// TwinCAT 3 PLC project CNM_Collections
// Title: CNM_Collections
// Company: ekvip automation GmbH
// Author: tdie
// ProjectVersion: 0.1.1.0
// Description: Concrete Implementations of Collections .. <legal notes> legal notes ================= | SPDX-FileCopyrightText: © 2024 ekvip automation GmbH <info@ekvip.de> | SPDX-License-Identifier: Apache-2.0 | For details check: Apache-2.0_ .. _Apache-2.0: https://www.apache.org/licenses/LICENSE-2.0 .. </legal notes>
// ProgramVersion: 3.1.4026.19
// libraries:
//   CNM_AbstractObject, * (ekvip automation GmbH)
//   CNM_CollectionInterfaces, * (ekvip automation GmbH)
//   CNM_CommandInterfaces, * (ekvip automation GmbH)
//   CNM_CycleManager, * (ekvip automation GmbH)
//   CNM_CycleManagerInterfaces, * (ekvip automation GmbH)
//   CNM_ReturnTypes, * (ekvip automation GmbH)
//   Tc2_System, * (Beckhoff Automation GmbH)
// project tree:
//   Appliers/classes/ ApplierBuilder.TcPOU, ApplierList.TcPOU, ChainedApplier.TcPOU
//   BinaryTree/BBSTIterator/classes/ AbstractBalancedBinarySearchTreeIterator.TcPOU, BfsBbstIterator.TcPOU, DfsBbstIterator.TcPOU, InorderBbstIterator.TcPOU
//   BinaryTree/BBSTIterator/interfaces/Iterator/ IBBSTIterator.TcIO
//   BinaryTree/classes/ BalancedBinarySearchTree.TcPOU, BalancedBinarySearchTreeNode.TcPOU
//   BinaryTree/Set/ InstantSetStrategyExecutor.TcPOU, SetStrategyExecutor.TcPOU
//   BinaryTree/Set/Interfaces/ ISetHelper.TcIO
//   BinaryTree/Tree/ InstantTreeStrategyExecutor.TcPOU, TreeStrategyExecutor.TcPOU
//   BinaryTree/Tree/Interfaces/ ITreeHelper.TcIO
//   Collection/classes/ AbstractCollection.TcPOU, AbstractDisposableContainer.TcPOU, ForEachStrategyExecutor.TcPOU, ForEachInstantStrategyExecutor.TcPOU
//   Factories/classes/ CollectionFactory.TcPOU
//   Iterate/classes/ AbstractIterator.TcPOU
//   Lists/ArrayList/ArrayListIterator/classes/ AbstractArrayListIterator.TcPOU, ForwardArrayListIterator.TcPOU, InverseArrayListIterator.TcPOU
//   Lists/ArrayList/ArrayListIterator/interfaces/Iterator/ IArrayListIterator.TcIO
//   Lists/ArrayList/ArrayListResizingStrategy/ CubicRootResizing.TcPOU, CubicRootUpsizeOnly.TcPOU
//   Lists/ArrayList/ArrayListSorter/ AbstractMergeBasedSorter.TcPOU, ArrayListMergeSorter.TcPOU, ArrayListShellSorter.TcPOU, ArrayListTwinSorter.TcPOU
//   Lists/ArrayList/classes/ ArrayList.TcPOU
//   Lists/ArrayList/ SortingOrder.TcDUT
//   Lists/classes/ AbstractList.TcPOU, SortingStrategyExecutor.TcPOU, InstantSortingStrategyExecutor.TcPOU
//   Lists/ IListHelpers.TcIO
//   Lists/LinkedList/classes/Interfaces/ ILinkedListHelpers.TcIO
//   Lists/LinkedList/classes/LinkedListIterator/classes/ AbstractLinkedListIterator.TcPOU, ForwardLinkedListIterator.TcPOU, InverseLinkedListIterator.TcPOU
//   Lists/LinkedList/classes/LinkedListIterator/interfaces/Iterator/ ILinkedListIterator.TcIO
//   Lists/LinkedList/classes/ DoublyLinkedElement.TcPOU, LinkedList.TcPOU
//   Lists/LinkedList/LinkedListSorter/ LinkedListMergeSorter.TcPOU
//   Lists/Sorter/classes/ AbstractArrayListSorter.TcPOU, AbstractLinkedListSorter.TcPOU, AbstractListSorter.TcPOU
//   Lists/Sorter/classes/Internal/ InvertComparator.TcPOU
//   Lists/Types/ IterationDirection.TcDUT
//   Parameter/ GeneralParameters.TcGVL
//   Project Information/ F_GetCompany.TcPOU, F_GetTitle.TcPOU, F_GetVersion.TcPOU
//   Utils/ FastSwap.TcPOU, log2.TcPOU
//   Version/ Global_Version.TcGVL

// ---- Lists/ArrayList/SortingOrder.TcDUT
{attribute 'qualified_only'}
{attribute 'strict'}
{attribute 'to_string'}
{attribute 'hide'}
TYPE FINAL SortingOrder :
(
	ASCENDING := 0,
	DESCENDING
) SINT;
END_TYPE

// ---- Lists/Types/IterationDirection.TcDUT
(*

## Short summary

This in an enumeration for the iteration direction. It can be forward (position) or backward (negative). 

.. <legal notes>

legal notes
=================
| SPDX-FileCopyrightText: © 2025 ekvip automation GmbH <info@ekvip.de>
| SPDX-License-Identifier: Apache-2.0
| For details check: Apache-2.0_

.. _Apache-2.0: https://www.apache.org/licenses/LICENSE-2.0

.. </legal notes>



*)

{attribute 'qualified_only'}
{attribute 'to_string'}
TYPE IterationDirection :
(
	BACKWARD := -1,
	FORWARD := 1
)DINT := FORWARD;
END_TYPE

// ---- Parameter/GeneralParameters.TcGVL
{attribute 'qualified_only'}
VAR_GLOBAL CONSTANT
	DEFAULT_OPERATIONS_PER_CYCLE :UDINT := 2048;
END_VAR

// ---- Version/Global_Version.TcGVL
{attribute 'TcGenerated'}
{attribute 'no-analysis'}
{attribute 'linkalways'}
// This function has been automatically generated from the project information.
VAR_GLOBAL CONSTANT
	{attribute 'const_non_replaced'}
	stLibVersion_CNM_Collections : ST_LibVersion := (iMajor := 0, iMinor := 1, iBuild := 1, iRevision := 0, nFlags := 0, sVersion := '0.1.1.0');
END_VAR

// ---- BinaryTree/BBSTIterator/interfaces/Iterator/IBBSTIterator.TcIO
(*

## Short summary

This interface extends the IIterator interface for collections by the method attachTree().

.. <legal notes>

legal notes
=================
| SPDX-FileCopyrightText: © 2022 ekvip automation GmbH <info@ekvip.de>
| SPDX-License-Identifier: Apache-2.0
| For details check: Apache-2.0_

.. _Apache-2.0: https://www.apache.org/licenses/LICENSE-2.0

.. </legal notes>

*)

INTERFACE IBBSTIterator EXTENDS CNM_CollectionInterfaces.IIterator

(*

## Short summary

This method attaches an binary balances search tree to the iterator.

.. <legal notes>

legal notes
=================
| SPDX-FileCopyrightText: © 2022 ekvip automation GmbH <info@ekvip.de>
| SPDX-License-Identifier: Apache-2.0
| For details check: Apache-2.0_

.. _Apache-2.0: https://www.apache.org/licenses/LICENSE-2.0

.. </legal notes>


*)

METHOD attachTree 
VAR_INPUT
	(* The tree to be attached, should not be NULL *)
	tree : REFERENCE TO BalancedBinarySearchTree;
END_VAR
END_METHOD

END_INTERFACE

// ---- BinaryTree/Set/Interfaces/ISetHelper.TcIO
INTERFACE INTERNAL ISetHelper EXTENDS CNM_AbstractObject.IObject

(*

## Short summary

Searches an object that is equal to the provided object in terms of the compareTo method (or a comparator provided by the parent).
 
.. <legal notes>

legal notes
=================
| SPDX-FileCopyrightText: © 2023 ekvip automation GmbH <info@ekvip.de>
| SPDX-License-Identifier: Apache-2.0
| For details check: Apache-2.0_

.. _Apache-2.0: https://www.apache.org/licenses/LICENSE-2.0

.. </legal notes>


**Return:** ``TRUE`` when an object that is equal is found, otherwise ``FALSE``

*)

METHOD INTERNAL getEqualObject :BOOL
VAR_INPUT
	(*The object to search for*)
	object 	:CNM_AbstractObject.IObject;
END_VAR
VAR_OUTPUT
	(*The found object or null if not found*)
	foundObject :CNM_AbstractObject.IObject;
END_VAR
END_METHOD

(*

## Short summary

overwrites the content of this set with the intersection of this set and the given set
Set intersection: Common elements between two sets.

**Example:**
Set A = {2, 3, 1, 4}
Set B = {3, 5, 6, 4}

Intersection of A and B: {3, 4}

.. <legal notes>

legal notes
=================
| SPDX-FileCopyrightText: © 2022 ekvip automation GmbH <info@ekvip.de>
| SPDX-License-Identifier: Apache-2.0
| For details check: Apache-2.0_

.. _Apache-2.0: https://www.apache.org/licenses/LICENSE-2.0

.. </legal notes>


**Return:** ``SingleExecutionResult.SUCCESS``: if intersect is complete
	``SingleExecutionResult.ABORTED``: foreign set wasn't valid

*)

METHOD INTERNAL instantIntersect :CNM_ReturnTypes.SingleExecutionResult
VAR_INPUT
	(*foreign set to intersect with*)
	set :CNM_CollectionInterfaces.ISet;
END_VAR
END_METHOD

(*

## Short summary

overwrites the content of this set with the union of this set and the given set
Set union: Combination of all elements from two sets.

**Example:**
Set A = {2, 3, 1, 4}
Set B = {3, 5, 6, 4}

Union of A and B: {1, 2, 3, 4, 5, 6}

.. <legal notes>

legal notes
=================
| SPDX-FileCopyrightText: © 2022 ekvip automation GmbH <info@ekvip.de>
| SPDX-License-Identifier: Apache-2.0
| For details check: Apache-2.0_

.. _Apache-2.0: https://www.apache.org/licenses/LICENSE-2.0

.. </legal notes>


**Return:** ``SUCCESS``: if merge completed
	```SingleExecutionResult.ABORTED``: foreign set wasn't valid

*)

METHOD INTERNAL instantMerge :CNM_ReturnTypes.SingleExecutionResult
VAR_INPUT
	(*foreign set to merge with*)
	set :CNM_CollectionInterfaces.ISet;
END_VAR
END_METHOD

(*

## Short summary

overwrites the content of this set with the set difference of this set and the given set
Set difference: Elements present in one set but not in the other.

**Example:**
Set A = {2, 3, 1, 4}
Set B = {3, 5, 6, 4}

Set difference (A - B): {1, 2}
Set difference (B - A): {5, 6}

.. <legal notes>

legal notes
=================
| SPDX-FileCopyrightText: © 2022 ekvip automation GmbH <info@ekvip.de>
| SPDX-License-Identifier: Apache-2.0
| For details check: Apache-2.0_

.. _Apache-2.0: https://www.apache.org/licenses/LICENSE-2.0

.. </legal notes>


**Return:** ``SingleExecutionResult.SUCCESS``: if insert could made, error if object was already in the tree,
	```SingleExecutionResult.ABORTED``: foreign set wasn't valid

*)

METHOD INTERNAL instantSubtract :CNM_ReturnTypes.SingleExecutionResult
VAR_INPUT
	(*foreign set to construct substraction*)
	set :CNM_CollectionInterfaces.ISet;
END_VAR
END_METHOD

(*

## Short summary

overwrites the content of this set with the intersection of this set and the given set
Set intersection: Common elements between two sets.

**Example:**
Set A = {2, 3, 1, 4}
Set B = {3, 5, 6, 4}

Intersection of A and B: {3, 4}

.. <legal notes>

legal notes
=================
| SPDX-FileCopyrightText: © 2022 ekvip automation GmbH <info@ekvip.de>
| SPDX-License-Identifier: Apache-2.0
| For details check: Apache-2.0_

.. _Apache-2.0: https://www.apache.org/licenses/LICENSE-2.0

.. </legal notes>


**Return:** ``SUCCESS``: if intersect is complete
	``ABORTED``: execute has a falling edge during intersect,
	``BUSY``: Intersect is in Progress
	``ERROR``: the passed collection was not valid / contained invalid Elements

*)

METHOD INTERNAL intersect :CNM_ReturnTypes.SingleExecutionState
VAR_INPUT
	(*foreign set to intersect with*)
	set :CNM_CollectionInterfaces.ISet;
	(*If intersect should be processed*)
	execute		:BOOL;
END_VAR
END_METHOD

(*

## Short summary

overwrites the content of this set with the union of this set and the given set
Set union: Combination of all elements from two sets.

**Example:**
Set A = {2, 3, 1, 4}
Set B = {3, 5, 6, 4}

Union of A and B: {1, 2, 3, 4, 5, 6}

.. <legal notes>

legal notes
=================
| SPDX-FileCopyrightText: © 2022 ekvip automation GmbH <info@ekvip.de>
| SPDX-License-Identifier: Apache-2.0
| For details check: Apache-2.0_

.. _Apache-2.0: https://www.apache.org/licenses/LICENSE-2.0

.. </legal notes>


**Return:** ``SUCCESS``: if merge completed, 
	``ABORTED``: execute has a falling edge during merge,
	``BUSY``: merge is in Progress
	``ERROR``: the passed collection where not valid / contained invalid Elements

*)

METHOD INTERNAL merge :CNM_ReturnTypes.SingleExecutionState
VAR_INPUT
	(*foreign set to merge with*)
	set :CNM_CollectionInterfaces.ISet;
	(*If merge should be processed*)
	execute		:BOOL;
END_VAR
END_METHOD

(*

## Short summary

overwrites the content of this set with the set difference of this set and the given set
Set difference: Elements present in one set but not in the other.

**Example:**
Set A = {2, 3, 1, 4}
Set B = {3, 5, 6, 4}

Set difference (A - B): {1, 2}
Set difference (B - A): {5, 6}

.. <legal notes>

legal notes
=================
| SPDX-FileCopyrightText: © 2022 ekvip automation GmbH <info@ekvip.de>
| SPDX-License-Identifier: Apache-2.0
| For details check: Apache-2.0_

.. _Apache-2.0: https://www.apache.org/licenses/LICENSE-2.0

.. </legal notes>


**Return:** ``SUCCESS``: if insert could made, error if object was already in the tree,
	``ABORTED``: execute has a falling edge during insert,
	``BUSY``: Insert is in Progress
	``ERROR``: the passed collection where not valid / contained invalid Elements

*)

METHOD INTERNAL subtract :CNM_ReturnTypes.SingleExecutionState
VAR_INPUT
	(*foreign set to construct substraction*)
	set :CNM_CollectionInterfaces.ISet;
	(*If substract should be processed*)
	execute		:BOOL;
END_VAR
END_METHOD

END_INTERFACE

// ---- BinaryTree/Tree/Interfaces/ITreeHelper.TcIO
INTERFACE INTERNAL ITreeHelper EXTENDS CNM_AbstractObject.IObject

(*

## Short summary

A method to insert a single element into the tree.

.. <legal notes>

legal notes
=================
| SPDX-FileCopyrightText: © 2022 ekvip automation GmbH <info@ekvip.de>
| SPDX-License-Identifier: Apache-2.0
| For details check: Apache-2.0_

.. _Apache-2.0: https://www.apache.org/licenses/LICENSE-2.0

.. </legal notes>


**Return:** ``SUCCESS``: operation successful
	``ABORTED``: operation was aborted (implementation specific)
	``ERROR``: out of memory

*)

METHOD INTERNAL insert :CNM_ReturnTypes.SingleExecutionResult
VAR_INPUT
	(*the object that should be inserted*)
	object :CNM_AbstractObject.IObject;
END_VAR
END_METHOD

(*

## Short summary

This method inserts all elements of a collection into the tree.

If any value of the collection could not be inserted because of duplication, operation isn't aborted, 
insertion is tried for every element of the collection.

.. <legal notes>

legal notes
=================
| SPDX-FileCopyrightText: © 2025 ekvip automation GmbH <info@ekvip.de>
| SPDX-License-Identifier: Apache-2.0
| For details check: Apache-2.0_

.. _Apache-2.0: https://www.apache.org/licenses/LICENSE-2.0

.. </legal notes>


**Return:** ``SUCCESS``: if insert could be made
	``ABORTED``: execute has a falling edge during insert,
	``BUSY``: Insert is in Progress
	``ERROR``: the passed collection where not valid / contained invalid Elements
	``IDLE``: method was never started

*)

METHOD INTERNAL insertCollection :CNM_ReturnTypes.SingleExecutionState
VAR_INPUT
	(*The collection that should be inserted*)
	collection	:CNM_CollectionInterfaces.ICollection;
	(*If insert should be processed*)
	execute		:BOOL;
END_VAR
END_METHOD

(*

## Short summary

This method inserts all elements of a collection into the tree
This takes only one cycle.

.. <legal notes>

legal notes
=================
| SPDX-FileCopyrightText: © 2022 ekvip automation GmbH <info@ekvip.de>
| SPDX-License-Identifier: Apache-2.0
| For details check: Apache-2.0_

.. _Apache-2.0: https://www.apache.org/licenses/LICENSE-2.0

.. </legal notes>


**Return:** ``SingleExecutionResult.SUCCESS``: operation successful
	``SingleExecutionResult.ERROR``: out of memory
	``SingleExecutionResult.ABORTED``: collection to insert wasn't valid

*)

METHOD INTERNAL instantInsertCollection :CNM_ReturnTypes.SingleExecutionResult
VAR_INPUT
	(*The collection that should be inserted*)
	collection	:CNM_CollectionInterfaces.ICollection;
END_VAR
END_METHOD

(*

## Short summary

Function to remove an object from the tree

.. <legal notes>

legal notes
=================
| SPDX-FileCopyrightText: © 2022 ekvip automation GmbH <info@ekvip.de>
| SPDX-License-Identifier: Apache-2.0
| For details check: Apache-2.0_

.. _Apache-2.0: https://www.apache.org/licenses/LICENSE-2.0

.. </legal notes>


**Return:** ``SUCCESS``: if remove could be made
	``ABORTED``: if object wasn't in the tree
	``ERROR``: if object wasn't valid

*)

METHOD INTERNAL remove :CNM_ReturnTypes.SingleExecutionResult
VAR_INPUT
	(* The object that should be removed *)
	object	:CNM_AbstractObject.IObject;
END_VAR
END_METHOD

END_INTERFACE

// ---- Lists/ArrayList/ArrayListIterator/interfaces/Iterator/IArrayListIterator.TcIO
(*

## Short summary

This interface extends the IIterator interface for collections by the method attachArrayList().

.. <legal notes>

legal notes
=================
| SPDX-FileCopyrightText: © 2022 ekvip automation GmbH <info@ekvip.de>
| SPDX-License-Identifier: Apache-2.0
| For details check: Apache-2.0_

.. _Apache-2.0: https://www.apache.org/licenses/LICENSE-2.0

.. </legal notes>

*)

INTERFACE IArrayListIterator EXTENDS CNM_CollectionInterfaces.IIterator

(*

## Short summary

This method attaches an array list to the iterator.

.. <legal notes>

legal notes
=================
| SPDX-FileCopyrightText: © 2024 ekvip automation GmbH <info@ekvip.de>
| SPDX-License-Identifier: Apache-2.0
| For details check: Apache-2.0_

.. _Apache-2.0: https://www.apache.org/licenses/LICENSE-2.0

.. </legal notes>

*)

METHOD attachArrayList
VAR_INPUT
	(* The list to be attached. Should be a reference of type ``ArrayList`` *)
	list :REFERENCE TO ArrayList;
END_VAR
END_METHOD

END_INTERFACE

// ---- Lists/IListHelpers.TcIO
INTERFACE INTERNAL IListHelpers EXTENDS CNM_CollectionInterfaces.IList

METHOD INTERNAL instantSorting : CNM_ReturnTypes.SingleExecutionResult
VAR_INPUT
	order :SortingOrder;
	(*Optional: the comparator that should be used for the sort. Must not be changed while sort is in process*)
	comparator	: CNM_CollectionInterfaces.CNM_AbstractObject.IComparator := 0;
END_VAR
END_METHOD

PROPERTY INTERNAL listChangeIndex : __XWORD
GET
END_GET
SET
END_SET
END_PROPERTY

METHOD INTERNAL sorting : CNM_ReturnTypes.SingleExecutionState
VAR_INPUT
	execute :BOOL;
	order :SortingOrder;
	(*Optional: the comparator that should be used for the sort. Must not be changed while sort is in process*)
	comparator	: CNM_CollectionInterfaces.CNM_AbstractObject.IComparator := 0;
END_VAR
END_METHOD

END_INTERFACE

// ---- Lists/LinkedList/classes/Interfaces/ILinkedListHelpers.TcIO
INTERFACE INTERNAL ILinkedListHelpers EXTENDS IListHelpers, CNM_CollectionInterfaces.ILinkedList

PROPERTY INTERNAL head : CNM_CollectionInterfaces.IDoublyLinkedElement
GET
END_GET
SET
END_SET
END_PROPERTY

PROPERTY INTERNAL last : CNM_CollectionInterfaces.IDoublyLinkedElement
GET
END_GET
SET
END_SET
END_PROPERTY

END_INTERFACE

// ---- Lists/LinkedList/classes/LinkedListIterator/interfaces/Iterator/ILinkedListIterator.TcIO
(*

## Short summary

This interface extends the IIterator interface for collections by the method attachLinkedList().

.. <legal notes>

legal notes
=================
| SPDX-FileCopyrightText: © 2022 ekvip automation GmbH <info@ekvip.de>
| SPDX-License-Identifier: Apache-2.0
| For details check: Apache-2.0_

.. _Apache-2.0: https://www.apache.org/licenses/LICENSE-2.0

.. </legal notes>

*)

INTERFACE ILinkedListIterator EXTENDS CNM_CollectionInterfaces.IIterator

(*

## Short summary

This method attaches an array list to the iterator.

.. <legal notes>

legal notes
=================
| SPDX-FileCopyrightText: © 2022 ekvip automation GmbH <info@ekvip.de>
| SPDX-License-Identifier: Apache-2.0
| For details check: Apache-2.0_

.. _Apache-2.0: https://www.apache.org/licenses/LICENSE-2.0

.. </legal notes>


**Return:** ``CNM_ReturnTypes.SingleExecutionResult.SUCCESS``: the list could be attached to the iterator

*)

METHOD attachLinkedList : CNM_ReturnTypes.SingleExecutionResult
VAR_INPUT
	(* The list to be attached. Should be of type ``CNM_CollectionInterfaces.ILinkedList`` *)
	list :REFERENCE TO LinkedList;
END_VAR
END_METHOD

END_INTERFACE

// ---- Appliers/classes/ApplierBuilder.TcPOU
FUNCTION_BLOCK ApplierBuilder EXTENDS AbstractDisposableContainer IMPLEMENTS CNM_CollectionInterfaces.IApplierChainBuilder, CNM_CollectionInterfaces.IApplierChainContinue
VAR
	applierList 		:ArrayList;
END_VAR

(*

## Short summary

Method to append another Applier to the chained applier.

.. <legal notes>

legal notes
=================
| SPDX-FileCopyrightText: © 2022 ekvip automation GmbH <info@ekvip.de>
| SPDX-License-Identifier: Apache-2.0
| For details check: Apache-2.0_

.. _Apache-2.0: https://www.apache.org/licenses/LICENSE-2.0

.. </legal notes>


**Return:** ``THIS^```IChainedApplier`

*)


METHOD andThen : CNM_CollectionInterfaces.IApplierChainContinue
VAR_INPUT
	applier :CNM_CollectionInterfaces.IApplier;
END_VAR
THIS^.applierList.append(applier);

andThen := THIS^;
END_METHOD

PROPERTY className : CNM_AbstractObject.ClassName
GET
className := 'ApplierBuilder';
END_GET
END_PROPERTY

(*

## Short summary

This method is called in the destruct method and is intended to zero all references and interfaces that should not be destructed. 
To delete the collection with all its contents, use deepDestruct() instead of destruct().

.. <legal notes>

legal notes
=================
| SPDX-FileCopyrightText: © 2025 ekvip automation GmbH <info@ekvip.de>
| SPDX-License-Identifier: Apache-2.0
| For details check: Apache-2.0_

.. _Apache-2.0: https://www.apache.org/licenses/LICENSE-2.0

.. </legal notes>

*)
METHOD PROTECTED clearContents
THIS^.applierList.clear();
END_METHOD

(*

## Short summary

Mark the object as deleted, as it stays in the memory.

.. <legal notes>

legal notes
=================
| SPDX-FileCopyrightText: © 2022 ekvip automation GmbH <info@ekvip.de>
| SPDX-License-Identifier: Apache-2.0
| For details check: Apache-2.0_

.. _Apache-2.0: https://www.apache.org/licenses/LICENSE-2.0

.. </legal notes>

*)
METHOD FB_Exit : BOOL
VAR_INPUT
	(* TRUE: the exit method is called in order to leave the instance which will be copied afterwards (online change).*)
	bInCopyCode	: BOOL;
END_VAR
IF THIS^.isObjectValid(THIS^.applierList) THEN
	THIS^.applierList.deepDestruct();
END_IF
END_METHOD

METHOD finish : CNM_CollectionInterfaces.IApplier
VAR
	object :CNM_AbstractObject.IObject;
	chainedApplier :POINTER TO ChainedApplier;
	applier1 :CNM_CollectionInterfaces.IApplier; 
	applier2 :CNM_CollectionInterfaces.IApplier; 
	applierNext :CNM_CollectionInterfaces.IApplier; 
END_VAR
IF(THIS^.applierList.size = 1)THEN
	__QUERYINTERFACE(THIS^.applierList.dequeue(), finish);
	THIS^.applierList.clear();
ELSE
	object := THIS^.applierList.dequeue();
	__QUERYINTERFACE(object, applier1);
	object := THIS^.applierList.dequeue();
	__QUERYINTERFACE(object, applier2);
	chainedApplier := __NEW(ChainedApplier(firstApplier := applier1, secondApplier := applier2));
	WHILE(THIS^.applierList.size > 0)DO
	object := THIS^.applierList.dequeue();
		__QUERYINTERFACE(object, applierNext);
		chainedApplier^.andThen(applierNext);
	END_WHILE
	finish := chainedApplier^;
END_IF
END_METHOD

METHOD startWith : CNM_CollectionInterfaces.IApplierChainContinue
VAR_INPUT
	applier :CNM_CollectionInterfaces.IApplier;
END_VAR
THIS^.applierList.clear();
THIS^.applierList.append(applier);

startWith := THIS^;
END_METHOD

END_FUNCTION_BLOCK

// ---- Collection/classes/AbstractDisposableContainer.TcPOU
(*

## Short summary

An abstract class to encapsulate 'destruct','deepDestruct' and 'fb_exit' logic.
'destructContents' must be implemented in the concrete class.

.. <legal notes>

legal notes
=================
| SPDX-FileCopyrightText: © 2025 ekvip automation GmbH <info@ekvip.de>
| SPDX-License-Identifier: Apache-2.0
| For details check: Apache-2.0_

.. _Apache-2.0: https://www.apache.org/licenses/LICENSE-2.0

.. </legal notes>



*)

FUNCTION_BLOCK ABSTRACT AbstractDisposableContainer EXTENDS CNM_AbstractObject.Object

(*

## Short summary

This method is called in the destruct method and is intended to zero all references and interfaces that should not be destructed. 
To delete the collection with all its contents, use deepDestruct() instead of destruct().

.. <legal notes>

legal notes
=================
| SPDX-FileCopyrightText: © 2025 ekvip automation GmbH <info@ekvip.de>
| SPDX-License-Identifier: Apache-2.0
| For details check: Apache-2.0_

.. _Apache-2.0: https://www.apache.org/licenses/LICENSE-2.0

.. </legal notes>

*)

METHOD PROTECTED ABSTRACT clearContents
END_METHOD

(*

## Short summary

This method is a self-destruction if the object was created dynamically.
If the object is a container class, the container content is destroyed with it.

**Attention:** 
	For derivations: **If a derived class needs ``deepDestruct`` this method must be overwritten.**
	otherwise it just calls `Object.destruct`. 


.. <legal notes>

legal notes
=================
| SPDX-FileCopyrightText: © 2022 ekvip automation GmbH <info@ekvip.de>
| SPDX-License-Identifier: Apache-2.0
| For details check: Apache-2.0_

.. _Apache-2.0: https://www.apache.org/licenses/LICENSE-2.0

.. </legal notes>

*)
METHOD deepDestruct
VAR
	(* __DELETE(THIS) is not allowed anymore in Tc 4026.
       tmp is just a helper pointer that points to this instance *)
	tmp : POINTER TO CNM_AbstractObject.Object;
END_VAR
IF (
	Tc2_System.F_CheckMemoryArea(pData := THIS, nSize := SIZEOF(THIS^))
	= Tc2_System.E_TcMemoryArea.Dynamic
) THEN
	tmp := THIS;
	__DELETE(tmp);
END_IF
END_METHOD

(*

## Short summary

This method is a self-destruction if the object was created dynamically.
The disposable container provides the option to clear contents that should not be deleted.

.. <legal notes>

legal notes
=================
| SPDX-FileCopyrightText: © 2025 ekvip automation GmbH <info@ekvip.de>
| SPDX-License-Identifier: Apache-2.0
| For details check: Apache-2.0_

.. _Apache-2.0: https://www.apache.org/licenses/LICENSE-2.0

.. </legal notes>

*)
METHOD FINAL destruct
VAR
	(* __DELETE(THIS) is not allowed anymore in Tc 4026.
       tmp is just a helper pointer that points to this instance *)
	tmp : POINTER TO CNM_AbstractObject.Object;
END_VAR
THIS^.clearContents();
SUPER^.destruct();
END_METHOD

END_FUNCTION_BLOCK

// ---- Appliers/classes/ApplierList.TcPOU
FUNCTION_BLOCK ApplierList 
EXTENDS AbstractDisposableContainer 
IMPLEMENTS CNM_CollectionInterfaces.IApplierList
VAR
	myList 				:ArrayList;
END_VAR

METHOD addApplier : CNM_ReturnTypes.SingleExecutionResult
VAR_INPUT
	applier :CNM_CollectionInterfaces.IApplier;
END_VAR
addApplier := THIS^.myList.append(applier);
END_METHOD

METHOD addAppliers : CNM_ReturnTypes.SingleExecutionResult
VAR_INPUT
	appliers :CNM_CollectionInterfaces.ICollection;
END_VAR
addAppliers := THIS^.myList.appendCollection(appliers);
END_METHOD

PROPERTY className : CNM_AbstractObject.ClassName
GET
className := 'ApplierList';
END_GET
END_PROPERTY

METHOD clear : BOOL
VAR_INPUT
END_VAR
THIS^.myList.clear();
END_METHOD

(*

## Short summary

This method is called in the destruct method and is intended to zero all references and interfaces that should not be destructed. 
To delete the collection with all its contents, use deepDestruct() instead of destruct().

.. <legal notes>

legal notes
=================
| SPDX-FileCopyrightText: © 2025 ekvip automation GmbH <info@ekvip.de>
| SPDX-License-Identifier: Apache-2.0
| For details check: Apache-2.0_

.. _Apache-2.0: https://www.apache.org/licenses/LICENSE-2.0

.. </legal notes>

*)
METHOD PROTECTED clearContents
THIS^.myList.clear();
END_METHOD

(*

## Short summary

This property returns the amount of appliers in the list

.. <legal notes>

legal notes
=================
| SPDX-FileCopyrightText: © 2024 ekvip automation GmbH <info@ekvip.de>
| SPDX-License-Identifier: Apache-2.0
| For details check: Apache-2.0_

.. _Apache-2.0: https://www.apache.org/licenses/LICENSE-2.0

.. </legal notes>

*)

PROPERTY count :UDINT
GET
count := THIS^.myList.size;
END_GET
END_PROPERTY

(*

## Short summary

Mark the object as deleted, as it staiys in the memory.

.. <legal notes>

legal notes
=================
| SPDX-FileCopyrightText: © 2022 ekvip automation GmbH <info@ekvip.de>
| SPDX-License-Identifier: Apache-2.0
| For details check: Apache-2.0_

.. _Apache-2.0: https://www.apache.org/licenses/LICENSE-2.0

.. </legal notes>

*)
METHOD FB_Exit : BOOL
VAR_INPUT
	(* TRUE: the exit method is called in order to leave the instance which will be copied afterwards (online change).*)
	bInCopyCode	: BOOL;
END_VAR
IF THIS^.isObjectValid(THIS^.myList) THEN
	THIS^.myList.deepDestruct();
END_IF
END_METHOD

(*

## Short summary

A method to get an applier at the given index.

.. <legal notes>

legal notes
=================
| SPDX-FileCopyrightText: © 2022 ekvip automation GmbH <info@ekvip.de>
| SPDX-License-Identifier: Apache-2.0
| For details check: Apache-2.0_

.. _Apache-2.0: https://www.apache.org/licenses/LICENSE-2.0

.. </legal notes>


**Return:** CNM_ReturnTypes.ExecutionState

*)

METHOD getApplier : CNM_CollectionInterfaces.IApplier
VAR_INPUT
	index	:UDINT;
END_VAR
VAR
	obj :CNM_AbstractObject.IObject;
END_VAR
THIS^.myList.getObjectAt(index := index, object => obj);
__TRY
	__QUERYINTERFACE(obj, getApplier);
__CATCH
	;
__ENDTRY
END_METHOD

PROPERTY list : CNM_CollectionInterfaces.IArrayList
GET
list := this^.myList;
END_GET
END_PROPERTY

END_FUNCTION_BLOCK

// ---- Lists/ArrayList/classes/ArrayList.TcPOU
(*

## Short summary

Implementation of IArrayList.
Does not allow null objects as data! Object is not null if isObjectValid is true.
Efficient if size stays small and index operations need to be performed in O(1).

**Warning:**
	Calling __DELETE directly on a Collection will bypass the destruct Context and therefore also delete the contained elements.

.. <legal notes>

legal notes
=================
| SPDX-FileCopyrightText: © 2022 ekvip automation GmbH <info@ekvip.de>
| SPDX-License-Identifier: Apache-2.0
| For details check: Apache-2.0_

.. _Apache-2.0: https://www.apache.org/licenses/LICENSE-2.0

.. </legal notes>



*)

{attribute 'enable_dynamic_creation'}
FUNCTION_BLOCK ArrayList EXTENDS AbstractList IMPLEMENTS CNM_CollectionInterfaces.IArrayList
VAR
	(*the container where the elements are stored*)
	container					:POINTER TO CNM_AbstractObject.IObject;
	(*how many space does the container has, NOT how many places are currently taken*)
	currentContainerCapacity	:UDINT;
	(*the sorter used to sort the list*) 
	injectedSorter				:CNM_CollectionInterfaces.IArrayListSorter;
	(*true if the sorter was created inside this list, false if set from outside*)
	privateSorter				:BOOL;
	(* injected resizing strategy *)
	injectedResizingStrategy :CNM_CollectionInterfaces.IResizingStrategy;
END_VAR

(*

## Short summary

This method is called every time the list changes and can notify other components.

.. <legal notes>

legal notes
=================
| SPDX-FileCopyrightText: © 2025 ekvip automation GmbH <info@ekvip.de>
| SPDX-License-Identifier: Apache-2.0
| For details check: Apache-2.0_

.. _Apache-2.0: https://www.apache.org/licenses/LICENSE-2.0

.. </legal notes>



*)

METHOD PROTECTED announceListChange
THIS^.changesToCollection := THIS^.changesToCollection+1;
END_METHOD

(*

## Short summary

This method adds the given object to the end of the list.
Adding NULL-Objects or THIS^ to the list is not possible.

.. <legal notes>

legal notes
=================
| SPDX-FileCopyrightText: © 2022 ekvip automation GmbH <info@ekvip.de>
| SPDX-License-Identifier: Apache-2.0
| For details check: Apache-2.0_

.. _Apache-2.0: https://www.apache.org/licenses/LICENSE-2.0

.. </legal notes>


**Return:** ``CNM_ReturnTypes.SingleExecutionResult.SUCCESS``: new Container could be allocated and data was copied
	``CNM_ReturnTypes.SingleExecutionResult.ERROR``: new Container couldn't be allocated, container left unchanged
	``CNM_ReturnTypes.SingleExecutionResult.ABORTED``: NULL object or the list itself was passed
	
*)
METHOD append :CNM_ReturnTypes.SingleExecutionResult
VAR_INPUT
	(*The object to be appended*)
	object	:CNM_AbstractObject.IObject;
END_VAR
append := CNM_ReturnTypes.SingleExecutionResult.ABORTED;
RETURN(THIS^.isEqual(object) OR_ELSE THIS^.isObjectNull(object));

append :=  THIS^.upscaleContainer(1); 
RETURN(append <> CNM_ReturnTypes.SingleExecutionResult.SUCCESS);
THIS^.container[THIS^.size] := object;
THIS^.incrementSize();
THIS^.announceListChange();
END_METHOD

(*

## Short summary

This method adds all elements of the given collection to the end of this list.

.. <legal notes>

legal notes
=================
| SPDX-FileCopyrightText: © 2025 ekvip automation GmbH <info@ekvip.de>
| SPDX-License-Identifier: Apache-2.0
| For details check: Apache-2.0_

.. _Apache-2.0: https://www.apache.org/licenses/LICENSE-2.0

.. </legal notes>


**Return:** ``CNM_ReturnTypes.SingleExecutionResult.SUCCESS``: new Container not needed / could be allocated and data was copied
	``CNM_ReturnTypes.SingleExecutionResult.ERROR``: new Container couldn't be allocated, container left unchanged
	``CNM_ReturnTypes.SingleExecutionResult.ABORTED``: NULL object or the list itself was passed

*)

METHOD appendCollection :CNM_ReturnTypes.SingleExecutionResult
VAR_INPUT
	(*The collection to be appended*)
	collectionToAppend		:CNM_CollectionInterfaces.ICollection;
END_VAR
VAR
	currentIndex 			:UDINT := 0;
	currentObject 			:CNM_AbstractObject.IObject;
	iterator				:CNM_CollectionInterfaces.IIterator;
	arrayListToAppend		:POINTER TO ArrayList;
	newContainer			:POINTER TO CNM_AbstractObject.IObject;
	newContainerSize 		:UDINT;
END_VAR
VAR CONSTANT
	REGISTER_SIZE :UDINT := SIZEOF(__XWORD);
END_VAR
appendCollection := CNM_ReturnTypes.SingleExecutionResult.ABORTED;
RETURN(THIS^.isObjectNull(collectionToAppend) OR_ELSE THIS^.isEqual(collectionToAppend));
appendCollection := CNM_ReturnTypes.SingleExecutionResult.SUCCESS;
RETURN (collectionToAppend.size = 0);
appendCollection := CNM_ReturnTypes.SingleExecutionResult.ERROR;
THIS^.resizingStrategy.getUpscaledCapacity(requestedSize := THIS^.size + collectionToAppend.size, currentCapacity := THIS^.currentContainerCapacity, newCapacity => newContainerSize);
newContainer := __NEW(__XWORD, newContainerSize);
RETURN(newContainer = 0);
IF (THIS^.size > 0) AND_THEN (Tc2_System.MEMMOVE(newContainer, THIS^.container, THIS^.size * REGISTER_SIZE) = 0) THEN
	__DELETE(newContainer);
	RETURN;
END_IF
IF (__QUERYPOINTER(collectionToAppend, arrayListToAppend)) THEN
	IF (Tc2_System.MEMMOVE(ADR(newContainer[THIS^.size]), arrayListToAppend^.container, collectionToAppend.size*REGISTER_SIZE) = 0) THEN
		__DELETE(newContainer);
		RETURN;
	END_IF
ELSE
	IF (collectionToAppend.createNewIterator(iterator => iterator) <> CNM_ReturnTypes.SingleExecutionResult.SUCCESS) THEN
		__DELETE(newContainer); 
		RETURN;
	END_IF
	
	iterator.iterate(execute := FALSE);
	WHILE (
		iterator.iterate(execute := TRUE, object => currentObject) 
		= CNM_ReturnTypes.SingleExecutionState.BUSY
	) DO
		newContainer[THIS^.size + currentIndex] := currentObject;
		currentIndex := (currentIndex + 1);
	END_WHILE
	iterator.destruct();
	IF (currentIndex < collectionToAppend.size) THEN
		__DELETE(newContainer); 
		RETURN;
	END_IF
END_IF
__DELETE(THIS^.container);
THIS^.container := newContainer;
THIS^.currentContainerCapacity := newContainerSize;
THIS^.incrementSize(collectionToAppend.size);
THIS^.announceListChange();
appendCollection := CNM_ReturnTypes.SingleExecutionResult.SUCCESS;
END_METHOD

(*

## Short summary

This abstract property returns the class name of the concrete object, 
which is useful to check the class name for ``__DELETE``.

.. <legal notes>

legal notes
=================
| SPDX-FileCopyrightText: © 2022 ekvip automation GmbH <info@ekvip.de>
| SPDX-License-Identifier: Apache-2.0
| For details check: Apache-2.0_

.. _Apache-2.0: https://www.apache.org/licenses/LICENSE-2.0

.. </legal notes>

*)
PROPERTY className : CNM_AbstractObject.ClassName
GET
className := 'CNM_Collections.ArrayList';
END_GET
END_PROPERTY

(*

## Short summary

This method clears/deletes all clearable data from this object.

.. <legal notes>

legal notes
=================
| SPDX-FileCopyrightText: © 2022 ekvip automation GmbH <info@ekvip.de>
| SPDX-License-Identifier: Apache-2.0
| For details check: Apache-2.0_

.. _Apache-2.0: https://www.apache.org/licenses/LICENSE-2.0

.. </legal notes>



*)

METHOD clear
__DELETE(THIS^.container);
THIS^.container := __NEW(__XWORD, 10);	

THIS^.collectionSize := 0;
THIS^.currentContainerCapacity := 10;
END_METHOD

(*

## Short summary

This method is called in the destruct method and is intended to zero all references and interfaces that should not be destructed. 
To delete the collection with all its contents, use deepDestruct() instead of destruct().

.. <legal notes>

legal notes
=================
| SPDX-FileCopyrightText: © 2025 ekvip automation GmbH <info@ekvip.de>
| SPDX-License-Identifier: Apache-2.0
| For details check: Apache-2.0_

.. _Apache-2.0: https://www.apache.org/licenses/LICENSE-2.0

.. </legal notes>

*)

METHOD PROTECTED clearContents
VAR CONSTANT
	(* NULL is a constant which is always 0 *)
	NULL				:__XWORD := 0;
END_VAR
Tc2_System.MEMSET(THIS^.container, 0, THIS^.size * SIZEOF(__XWORD));
THIS^.injectedSorter := 0;
THIS^.injectedResizingStrategy := 0;
END_METHOD

(*

## Short summary

This method is used to create a new instance
of the object which has the same internal state as the object.
If the object is a container class, the references to the content objects
are not cloned for this there is the method `ICloneable.deepClone`.

If an object does not support cloning the return value is
``CNM_ReturnTypes.CloneResult.CLONE_IS_NOT_SUPPORTED``.

If there is not enough memory or the cloning fails because the
attribute enable dynamic creation was forgotten the return value is 
``CNM_ReturnTypes.CloneResult.FAILED``.

Only if the return value is ``CNM_ReturnTypes.CloneResult.SUCCESS``
the output ``clonedObject`` points to the new object
otherwise ``clonedObject`` is NULL.  

**Attention:** 
	For derivations: **If a derived class needs ``clone`` this method must be overwritten.**
	and don't forget the attribute ``{attribute 'enable_dynamic_creation'}``  

.. <legal notes>

legal notes
=================
| SPDX-FileCopyrightText: © 2022 ekvip automation GmbH <info@ekvip.de>
| SPDX-License-Identifier: Apache-2.0
| For details check: Apache-2.0_

.. _Apache-2.0: https://www.apache.org/licenses/LICENSE-2.0

.. </legal notes>


**Return:**``CNM_ReturnTypes.CloneResult.SUCCESS``: new object clone was created,
``CNM_ReturnTypes.CloneResult.FAILED``: object clone failed
``CNM_ReturnTypes.CloneResult.CLONE_IS_NOT_SUPPORTED``: object does not support cloning

*)
METHOD clone : CNM_AbstractObject.CNM_ReturnTypes.CloneResult
VAR_OUTPUT
	(* new object instance or NULL if somthing went wrong *)
	clonedObject	:CNM_AbstractObject.IObject;
END_VAR
VAR
	result :CNM_ReturnTypes.SingleExecutionResult;
	miniMe :POINTER TO ArrayList;
END_VAR
clone := CNM_ReturnTypes.CloneResult.FAILED;
miniMe := __NEW(ArrayList);
RETURN (miniMe = 0);
clone := CNM_ReturnTypes.CloneResult.SUCCESS;
clonedObject := miniMe^;
IF (miniMe^.appendCollection(THIS^) <> CNM_ReturnTypes.SingleExecutionResult.SUCCESS) THEN
	clonedObject.destruct();
	clone := CNM_ReturnTypes.CloneResult.FAILED;
	clonedObject := 0;
END_IF
END_METHOD

(*

## Short summary

This method returns a NEW Iterator instance which can iterate the collection.
These iterators can be used parallel independend of each other on the same collection.

**Warning:**
The returned Iterator was created using the __NEW operator and must be destructed to avoid memory leaks!



.. <legal notes>

legal notes
=================
| SPDX-FileCopyrightText: © 2024 ekvip automation GmbH <info@ekvip.de>
| SPDX-License-Identifier: Apache-2.0
| For details check: Apache-2.0_

.. _Apache-2.0: https://www.apache.org/licenses/LICENSE-2.0

.. </legal notes>



*)

METHOD createNewIterator :CNM_CollectionInterfaces.CNM_ReturnTypes.SingleExecutionResult
VAR_OUTPUT
	(*The new created iterator or null if allocation fails *)
	iterator	:CNM_CollectionInterfaces.IIterator;
END_VAR
VAR
	newIterator :POINTER TO ForwardArrayListIterator;
END_VAR
newIterator := __NEW(ForwardArrayListIterator(arrayList := THIS^));
IF (newIterator = 0) THEN
	createNewIterator := CNM_ReturnTypes.SingleExecutionResult.ERROR;
	RETURN;
END_IF
createNewIterator := CNM_ReturnTypes.SingleExecutionResult.SUCCESS;
iterator := newIterator^;
END_METHOD

(*

## Short summary

reduces the collection size by the number of removed elements.

.. <legal notes>

legal notes
=================
| SPDX-FileCopyrightText: © 2025 ekvip automation GmbH <info@ekvip.de>
| SPDX-License-Identifier: Apache-2.0
| For details check: Apache-2.0_

.. _Apache-2.0: https://www.apache.org/licenses/LICENSE-2.0

.. </legal notes>

*)

METHOD PROTECTED decrementSize
VAR_INPUT
	numberOfRemovedElements :UDINT := 1;
END_VAR
THIS^.collectionSize := THIS^.collectionSize - numberOfRemovedElements;
END_METHOD

(*

## Short summary

This method is used to create a new instance
of the object which has the same internal state as the object.
If the object is a container class, the references to the content objects
are cloned too.

If an object does not support cloning the return value is
``CNM_ReturnTypes.CloneResult.CLONE_IS_NOT_SUPPORTED``.

If there is not enough memory or the cloning fails because the
attribute enable dynamic creation was forgotten the return value is 
``CNM_ReturnTypes.CloneResult.FAILED``.
If something goes wrong, then this method must clean up everything
that has been cloned and free the memory again.
**The deepClone either works completely, or not at all**

Only if the return value is ``CNM_ReturnTypes.CloneResult.SUCCESS``
the output ``clonedObject`` points to the new object
otherwise ``clonedObject`` is NULL.  

**Attention:** 
	For derivations: **If a derived class needs ``deepClone`` this method must be overwritten.**
	and don't forget the attribute ``{attribute 'enable_dynamic_creation'}``, even for container content 

.. <legal notes>

legal notes
=================
| SPDX-FileCopyrightText: © 2022 ekvip automation GmbH <info@ekvip.de>
| SPDX-License-Identifier: Apache-2.0
| For details check: Apache-2.0_

.. _Apache-2.0: https://www.apache.org/licenses/LICENSE-2.0

.. </legal notes>


**Return:**``CNM_ReturnTypes.CloneResult.SUCCESS``: new object clone was created,
``CNM_ReturnTypes.CloneResult.FAILED``: object clone failed
``CNM_ReturnTypes.CloneResult.CLONE_IS_NOT_SUPPORTED``: object does not support deep cloning

*)
METHOD deepClone : CNM_AbstractObject.CNM_ReturnTypes.CloneResult
VAR_OUTPUT
	(* new object instance or NULL if somthing went wrong *)
	clonedObject	: CNM_AbstractObject.IObject;
END_VAR
VAR
	result :CNM_ReturnTypes.SingleExecutionResult;
	miniMe :POINTER TO ArrayList;
	newInstance :CNM_CollectionInterfaces.IArrayList;
	clonedSorter :CNM_CollectionInterfaces.IArrayListSorter;
	clonedSorterObject :CNM_AbstractObject.IObject;
	index :UDINT;
	target :UDINT;
	tmpObject :CNM_AbstractObject.IObject;
	currentObject :CNM_AbstractObject.IObject;
END_VAR
deepClone := CNM_ReturnTypes.CloneResult.FAILED;
miniMe := __NEW(ArrayList);
RETURN (miniMe = 0);
deepClone := CNM_ReturnTypes.CloneResult.SUCCESS;
clonedObject := miniMe^;
newInstance := miniMe^;
IF (THIS^.size > 0) THEN
	target := THIS^.size - 1;
	FOR index := 0 TO target DO
		currentObject := THIS^.container[index];
		IF NOT THIS^.isObjectValid(currentObject) THEN
			deepClone := CNM_ReturnTypes.CloneResult.FAILED;
			miniMe^.deepDestruct();
			clonedObject := 0;
			RETURN;
		ELSE 
			deepClone := currentObject.deepClone(clonedObject => tmpObject);
			IF (deepClone <> CNM_ReturnTypes.CloneResult.SUCCESS) THEN 
				miniMe^.deepDestruct();
				clonedObject := 0;
				RETURN;
			END_IF
			IF (miniMe^.append(tmpObject) <> CNM_ReturnTypes.SingleExecutionResult.SUCCESS) THEN
				deepClone := CNM_ReturnTypes.CloneResult.FAILED;
				miniMe^.deepDestruct();
				clonedObject := 0;
				RETURN;
			END_IF
		END_IF
	END_FOR
END_IF
	
RETURN (THIS^.isObjectNull(THIS^.injectedSorter));
THIS^.injectedSorter.deepClone(clonedObject => clonedSorterObject);
__QUERYINTERFACE(clonedSorterObject, clonedSorter);
deepClone := SEL(
	THIS^.isObjectValid(clonedSorter),
	CNM_ReturnTypes.CloneResult.FAILED,
	CNM_ReturnTypes.CloneResult.SUCCESS
);

IF (THIS^.isObjectNull(clonedSorter)) THEN
	deepClone := CNM_ReturnTypes.CloneResult.FAILED;
	miniMe^.deepDestruct();
	clonedObject := 0;
	RETURN;
END_IF
newInstance.setSorter(sorter := clonedSorter);
END_METHOD

(*

## Short summary

This property returns the first object in the list and removes it from the list. 
Can be seen as opposite of prepend.
**Example:**
On a list: (Head -->) A B C, list.dequeue will return A.
**Example 2:**
If you call prepend(x), a dequeue right after will return x.

.. <legal notes>

legal notes
=================
| SPDX-FileCopyrightText: © 2022 ekvip automation GmbH <info@ekvip.de>
| SPDX-License-Identifier: Apache-2.0
| For details check: Apache-2.0_

.. _Apache-2.0: https://www.apache.org/licenses/LICENSE-2.0

.. </legal notes>



*)

METHOD dequeue :CNM_AbstractObject.IObject
VAR CONSTANT
	NULL_REFERENCE :__XWORD := 0;
END_VAR
IF (THIS^.size = 0) THEN
	dequeue := NULL_REFERENCE;
	RETURN;
END_IF
dequeue := THIS^.container[0];
THIS^.leftShiftObjects(1);
THIS^.decrementSize();
THIS^.downscaleContainer();
THIS^.announceListChange();
END_METHOD

(*

## Short summary

This method is called in the deepDestruct method and is intended to destruct all contained Objects of the collection. 
To delete only the collection without deleting all its contents, use destruct() instead of deepDestruct().

.. <legal notes>

legal notes
=================
| SPDX-FileCopyrightText: © 2025 ekvip automation GmbH <info@ekvip.de>
| SPDX-License-Identifier: Apache-2.0
| For details check: Apache-2.0_

.. _Apache-2.0: https://www.apache.org/licenses/LICENSE-2.0

.. </legal notes>

*)

METHOD PROTECTED destructContents
VAR
	currentIndex	:__XWORD;
END_VAR
IF (container <> 0) THEN
	FOR currentIndex := 0 TO (THIS^.currentContainerCapacity - 1) DO
		IF THIS^.isObjectValid(THIS^.container[currentIndex]) THEN
			THIS^.container[currentIndex].deepDestruct();
		END_IF
	END_FOR
END_IF
END_METHOD

(*

## Short summary

This method decreases the container capacity by the current decrease strategy amount.

.. <legal notes>

legal notes
=================
| SPDX-FileCopyrightText: © 2025 ekvip automation GmbH <info@ekvip.de>
| SPDX-License-Identifier: Apache-2.0
| For details check: Apache-2.0_

.. _Apache-2.0: https://www.apache.org/licenses/LICENSE-2.0

.. </legal notes>


**Return:** ``CNM_ReturnTypes.SingleExecutionResult.SUCCESS``: new Container could be allocated and data was copied
	``CNM_ReturnTypes.SingleExecutionResult.ERROR``: new Container couldn't be allocated, container left unchanged

*)

{info 'add logging if containeralloc fails'}
METHOD PROTECTED downscaleContainer :CNM_ReturnTypes.SingleExecutionResult;
VAR
	newContainer 			:POINTER TO CNM_AbstractObject.IObject;
	lastContainerCapacity	:UDINT;
	newContainerCapacity	:UDINT;
END_VAR
IF THIS^.resizingStrategy.getDownscaledCapacity(
		requestedSize := THIS^.size,
		currentCapacity := THIS^.currentContainerCapacity,
		newCapacity => newContainerCapacity
	)
THEN
	newContainer := __NEW(__XWORD, newContainerCapacity);
	IF (newContainer <> 0) THEN
		IF (THIS^.container <> 0) THEN 
			IF (THIS^.size > 0) THEN
				Tc2_System.MEMCPY(newContainer, THIS^.container,  THIS^.size * SIZEOF(__XWORD));
			END_IF
			__DELETE(THIS^.container);
		END_IF
		THIS^.container := newContainer;
		downscaleContainer := CNM_ReturnTypes.SingleExecutionResult.SUCCESS;
	ELSE
		THIS^.currentContainerCapacity := lastContainerCapacity;
		downscaleContainer := CNM_ReturnTypes.SingleExecutionResult.ERROR;
	END_IF
END_IF
END_METHOD

(*

## Short summary

Mark the object as deleted, as it staiys in the memory.

.. <legal notes>

legal notes
=================
| SPDX-FileCopyrightText: © 2022 ekvip automation GmbH <info@ekvip.de>
| SPDX-License-Identifier: Apache-2.0
| For details check: Apache-2.0_

.. _Apache-2.0: https://www.apache.org/licenses/LICENSE-2.0

.. </legal notes>

*)
METHOD FB_Exit : BOOL
VAR_INPUT
	(* TRUE: the exit method is called in order to leave the instance which will be copied afterwards (online change).*)
	bInCopyCode	: BOOL;
END_VAR
VAR
	currentIndex	:__XWORD;
END_VAR
IF (container <> 0) THEN
	FOR currentIndex := 0 TO (THIS^.currentContainerCapacity - 1) DO
		IF THIS^.isObjectValid(THIS^.container[currentIndex]) THEN
			THIS^.container[currentIndex].deepDestruct();
		END_IF
	END_FOR
END_IF
IF (THIS^.container <> 0) THEN
	__DELETE(container);
END_IF
IF THIS^.isObjectValid(THIS^.injectedSorter) THEN
	 THIS^.injectedSorter.deepDestruct();
END_IF
IF THIS^.isObjectValid(THIS^.injectedResizingStrategy) THEN
	THIS^.injectedResizingStrategy.deepDestruct();
END_IF
END_METHOD

(*

## Short summary

This method returns the index of the first object that is equal to the given object.

.. <legal notes>

legal notes
=================
| SPDX-FileCopyrightText: © 2022 ekvip automation GmbH <info@ekvip.de>
| SPDX-License-Identifier: Apache-2.0
| For details check: Apache-2.0_

.. _Apache-2.0: https://www.apache.org/licenses/LICENSE-2.0

.. </legal notes>


**Return:** ``CNM_ReturnTypes.SingleExecutionResult.SUCCESS``: Element was found inside the list
	``CNM_ReturnTypes.SingleExecutionResult.ERROR``: object could not be found in the list
	
*)

METHOD getIndexOf : CNM_ReturnTypes.SingleExecutionResult
VAR_INPUT
	(*the object to get the index from*)
	object	:CNM_AbstractObject.IObject;
END_VAR
VAR_OUTPUT
	(*The index where the first occurence was found, only valid if return value was SUCCESS, else undefined(UDINT#FFFF_FFFF) *)
	index	:UDINT;
END_VAR
VAR
	currentObject 	:CNM_AbstractObject.IObject;
END_VAR
THIS^.iterate(FALSE);
IF (THIS^.isObjectValid(object)) THEN
	WHILE (
		THIS^.iterate(execute := TRUE, object => currentObject) 
		= CNM_ReturnTypes.SingleExecutionState.BUSY
	) DO
		IF (object.isEqual(currentObject)) THEN
			getIndexOf := CNM_ReturnTypes.SingleExecutionResult.SUCCESS;
			RETURN;
		END_IF
		index := index +1;
	END_WHILE
END_IF

//in case of not found set index to UDINT max 
index := UDINT#16#FFFF_FFFF;
getIndexOf := CNM_ReturnTypes.SingleExecutionResult.ERROR;
END_METHOD

(*

## Short summary

This method returns the object at the given index.

.. <legal notes>

legal notes
=================
| SPDX-FileCopyrightText: © 2022 ekvip automation GmbH <info@ekvip.de>
| SPDX-License-Identifier: Apache-2.0
| For details check: Apache-2.0_

.. _Apache-2.0: https://www.apache.org/licenses/LICENSE-2.0

.. </legal notes>


**Return:** ``CNM_ReturnTypes.SingleExecutionResult.SUCCESS``: index within valid range, object could be retrieved
	``CNM_ReturnTypes.SingleExecutionResult.ERROR``: index was out of valid range

*)

METHOD getObjectAt : CNM_ReturnTypes.SingleExecutionResult
VAR_INPUT
	(*the index to access the object from*)
	index	:UDINT;
END_VAR
VAR_OUTPUT
	(*The object found at the index, undefined if ERROR*)
	object	: CNM_AbstractObject.IObject;
END_VAR
VAR CONSTANT
	NULL_REFERENCE :__XWORD := 0;
END_VAR
IF (index >= THIS^.size) THEN
	getObjectAt := CNM_ReturnTypes.SingleExecutionResult.ERROR;
	object := NULL_REFERENCE;
	RETURN;
END_IF

getObjectAt := CNM_ReturnTypes.SingleExecutionResult.SUCCESS;
object := THIS^.container[index];
END_METHOD

(*

## Short summary

Increments the collectionsize by given amount. 

.. <legal notes>

legal notes
=================
| SPDX-FileCopyrightText: © 2025 ekvip automation GmbH <info@ekvip.de>
| SPDX-License-Identifier: Apache-2.0
| For details check: Apache-2.0_

.. _Apache-2.0: https://www.apache.org/licenses/LICENSE-2.0

.. </legal notes>

*)

METHOD PROTECTED incrementSize
VAR_INPUT
	numberOfAddedElements :UDINT := 1;
END_VAR
THIS^.collectionSize := (THIS^.collectionSize + numberOfAddedElements);
END_METHOD

(*

## Short summary

This method inserts the given object at the given index. 
The element that was on this index before is not deleted,
but instead is shifted right by one position together 
with the other elements on indices larger than ``index``.
If ``object`` is not valid, list is left unchanged.

.. <legal notes>

legal notes
=================
| SPDX-FileCopyrightText: © 2022 ekvip automation GmbH <info@ekvip.de>
| SPDX-License-Identifier: Apache-2.0
| For details check: Apache-2.0_

.. _Apache-2.0: https://www.apache.org/licenses/LICENSE-2.0

.. </legal notes>


**Return:** ``CNM_ReturnTypes.SingleExecutionResult.SUCCESS``: insert was successful
	``CNM_ReturnTypes.SingleExecutionResult.ERROR``: insert failed, because container needs to increase but no memory left or index is not in valid range
	``CNM_ReturnTypes.SingleExecutionResult.ABORTED``: NULL object or the list itself was passed
*)

METHOD insertObjectAt :CNM_ReturnTypes.SingleExecutionResult
VAR_INPUT
	(*the index to insert the object at*)
	index	:UDINT;
	(*the object to be inserted*)
	object	:CNM_AbstractObject.IObject;
END_VAR
insertObjectAt := CNM_ReturnTypes.SingleExecutionResult.ABORTED;
RETURN(THIS^.isObjectNull(object) OR_ELSE THIS^.isEqual(object));
insertObjectAt := CNM_ReturnTypes.SingleExecutionResult.ERROR;
RETURN (index > THIS^.size);

IF THIS^.isObjectValid(object) THEN
	THIS^.upscaleContainer(1);
	IF (THIS^.rightShiftObjects(index) <> CNM_ReturnTypes.SingleExecutionResult.SUCCESS) THEN
		THIS^.downscaleContainer();
		RETURN;
	END_IF
	THIS^.container[index] := object;
	THIS^.incrementSize();
	THIS^.announceListChange();
	insertObjectAt := CNM_ReturnTypes.SingleExecutionResult.SUCCESS;
END_IF
END_METHOD

METHOD INTERNAL instantSorting : CNM_ReturnTypes.SingleExecutionResult
VAR_INPUT
	order :SortingOrder;
	(*Optional: the comparator that should be used for the sort. Must not be changed while sort is in process*)
	comparator	: CNM_CollectionInterfaces.CNM_AbstractObject.IComparator := 0;
END_VAR
CASE order OF
SortingOrder.ASCENDING:
	instantSorting := THIS^.sorter.instantSort(
		size := THIS^.size, 
		comparator := comparator, 
		container := THIS^.container, 
		currentListVersion := THIS^.changesToCollection
	);

SortingOrder.DESCENDING:
	instantSorting	:= THIS^.sorter.instantInverseSort(
		size := THIS^.size, 
		container := THIS^.container, 
		currentListVersion := THIS^.changesToCollection
	);
	
END_CASE
END_METHOD


(*

## Short summary

Inverts the order of the elements inside the list. 
Does not apply any kind of sorting, only reverses the elements in the list.

.. <legal notes>

legal notes
=================
| SPDX-FileCopyrightText: © 2022 ekvip automation GmbH <info@ekvip.de>
| SPDX-License-Identifier: Apache-2.0
| For details check: Apache-2.0_

.. _Apache-2.0: https://www.apache.org/licenses/LICENSE-2.0

.. </legal notes>

*)

METHOD invert
VAR
	firstElement	:UDINT := 0;
	lastElement		:UDINT := THIS^.size - 1;
	midLower		:UDINT;
	midUpper		:UDINT;
	loop			:UDINT;
END_VAR
VAR CONSTANT
	REGISTER_SIZE :__XWORD := SIZEOF(__XWORD);
END_VAR
CASE (THIS^.size) OF
0,1: RETURN;
2,3: FastSwap(ADR(THIS^.container[firstElement]), ADR(THIS^.container[lastElement]));RETURN;
ELSE
	loop := SHR(THIS^.size, 1);
	midLower := loop - 1;
	midUpper := THIS^.size - loop;
	
	IF ((loop AND 1) <> 0) THEN
		FastSwap(ADR(THIS^.container[midLower]), ADR(THIS^.container[midUpper]));
		loop := loop - 1;
		midLower := midLower - 1;
		midUpper := midupper + 1;
	END_IF;
	
	loop := MAX(SHR(loop, 1), 1);	
END_CASE
	
REPEAT
	FastSwap(ADR(THIS^.container[firstElement]),ADR(THIS^.container[lastElement]));	
	FastSwap(ADR(THIS^.container[midLower]),ADR(THIS^.container[midUpper]));	
	midLower := midLower - 1;
	midUpper := midupper + 1;
	firstElement := firstElement + 1;
	lastElement := lastElement - 1; 
	loop := loop - 1;
UNTIL (loop = 0) END_REPEAT
END_METHOD

(*

## Short summary

This method returns the next object in the list and returns an execution state.

.. <legal notes>

legal notes
=================
| SPDX-FileCopyrightText: © 2022 ekvip automation GmbH <info@ekvip.de>
| SPDX-License-Identifier: Apache-2.0
| For details check: Apache-2.0_

.. _Apache-2.0: https://www.apache.org/licenses/LICENSE-2.0

.. </legal notes>


**Return:** ``SUCCESS``: if last object from collection was returned,
	``ABORTED``: execute has a falling edge during iterate,
	``BUSY``: When iterate had rising edge on execute and not all objects had been returned yet
	``IDLE``: iterate not in progress, execute is false and iterate reseted 

*)
METHOD PROTECTED iterate :CNM_ReturnTypes.SingleExecutionState
VAR_INPUT
	(*False to init, True to retrieve next element*)
	execute	: BOOL;
END_VAR
VAR_OUTPUT
	(*The current element of the iteration*)
	object	:CNM_AbstractObject.IObject;
END_VAR
VAR_INST
	lastExecute 	:BOOL;
	state 			:CNM_ReturnTypes.SingleExecutionState := CNM_ReturnTypes.SingleExecutionState.IDLE;
	currentIndex	:UDINT;
	cycleManager 	:CNM_CycleManager.SimpleCycleManager;
	currentListVersion :__XWORD;
END_VAR
VAR CONSTANT
	IS_NOT_REFERENCED 	:__XWORD := 0;	
	INIT 		:DINT := CNM_ReturnTypes.DefaultSteps.STEP.INIT;
	ITERATING 	:DINT := INIT +1;
	ERROR 		:DINT := CNM_ReturnTypes.DefaultSteps.STEP.ERROR;
END_VAR
IF (cycleManager.step.current > INIT) THEN
	cycleManager.assert.bitNumber.x.valueIsEqualTo(
		currentValue := currentListVersion,
		expectedValue := THIS^.changesToCollection,
		message := 'This instance of ArrayList has changed between iterate calls'
	);
END_IF

cycleManager(execute := execute);
CASE cycleManager.step.current OF
INIT:
	object := IS_NOT_REFERENCED;
	currentIndex := 0;
	currentListVersion := THIS^.changesToCollection;
	IF (currentIndex < THIS^.size) THEN
		object := THIS^.container[currentIndex];
		currentIndex := currentIndex + 1;
		cycleManager.proceed();
	ELSE
		cycleManager.proceedWith(CNM_ReturnTypes.DefaultSteps.STEP.SUCCESS);
		object := IS_NOT_REFERENCED;
	END_IF
ITERATING:
	IF (currentIndex < THIS^.size) THEN
		object := THIS^.container[currentIndex];
		currentIndex := currentIndex + 1;
	ELSE
		cycleManager.proceedWith(CNM_ReturnTypes.DefaultSteps.STEP.SUCCESS);
		object := IS_NOT_REFERENCED;
	END_IF
ERROR:
	object := IS_NOT_REFERENCED;
END_CASE

iterate := cycleManager.state;
END_METHOD

(*

## Short summary

This method shifts the data in the container to the left at the given index.
It memsets the free created gap at the end of the container.
leftShift(0) : A B C D -> B C D
leftShift(1) : A B C D -> A C D
leftShift(1, 2) : A B C D -> A D

.. <legal notes>

legal notes
=================
| SPDX-FileCopyrightText: © 2025 ekvip automation GmbH <info@ekvip.de>
| SPDX-License-Identifier: Apache-2.0
| For details check: Apache-2.0_

.. _Apache-2.0: https://www.apache.org/licenses/LICENSE-2.0

.. </legal notes>


**Return:** ``CNM_ReturnTypes.SingleExecutionResult.SUCCESS``: leftshift was successful
	``CNM_ReturnTypes.SingleExecutionResult.ERROR``: startindex was either zero ,less than distance or greater thansize, distance greater than size

*)

METHOD PROTECTED leftShiftObjects :CNM_ReturnTypes.SingleExecutionResult;
VAR_INPUT
	(*where the leftshift should start, position of the first element which will shift to the left. All elements after this are also shifted by the same amount.*)
	startIndex :UDINT;
	(* the size of the gap to be shifted to the left as IObjects *)
	distance :UDINT := 1;
END_VAR
VAR
	objectsToShift :UDINT;
END_VAR
VAR CONSTANT
	IS_NOT_REFERENCED 	:USINT := 0;
	REGISTER_SIZE :UDINT := SIZEOF(__XWORD);
END_VAR
leftShiftObjects := CNM_ReturnTypes.SingleExecutionResult.ERROR;
RETURN((distance >= THIS^.size) OR_ELSE (startIndex = 0) OR_ELSE (startIndex < distance) OR_ELSE (THIS^.size < startIndex));
objectsToShift := THIS^.size - startIndex;
Tc2_System.MEMMOVE(ADR(THIS^.container[startIndex-distance]), ADR(THIS^.container[startIndex]), objectsToShift * REGISTER_SIZE);
Tc2_System.MEMSET(ADR(THIS^.container[THIS^.size-distance]), IS_NOT_REFERENCED, distance * REGISTER_SIZE);
leftShiftObjects := CNM_ReturnTypes.SingleExecutionResult.SUCCESS;
END_METHOD

(*

## Short summary

This property returns the last object in the list and removes it from the list. 
Can be seen as opposite of append.
**Example:**
On a list: (Head -->) A B C, list.pop will return C.
**Example 2:**
If you call append(x), a pop right after will return x.

.. <legal notes>

legal notes
=================
| SPDX-FileCopyrightText: © 2022 ekvip automation GmbH <info@ekvip.de>
| SPDX-License-Identifier: Apache-2.0
| For details check: Apache-2.0_

.. _Apache-2.0: https://www.apache.org/licenses/LICENSE-2.0

.. </legal notes>



*)

METHOD pop :CNM_AbstractObject.IObject
VAR CONSTANT
	NULL_REFERENCE :__XWORD := 0;
END_VAR
IF (THIS^.size = 0) THEN
	pop := NULL_REFERENCE;
	RETURN;
END_IF
pop := THIS^.container[THIS^.size-1];
THIS^.container[THIS^.size-1] := NULL_REFERENCE;
THIS^.decrementSize();
THIS^.downscaleContainer();
THIS^.announceListChange();
END_METHOD

(*

## Short summary

This method adds the given object to the start of the list.
Adding NULL-Objects or THIS^ to the list is not possible.

.. <legal notes>

legal notes
=================
| SPDX-FileCopyrightText: © 2022 ekvip automation GmbH <info@ekvip.de>
| SPDX-License-Identifier: Apache-2.0
| For details check: Apache-2.0_

.. _Apache-2.0: https://www.apache.org/licenses/LICENSE-2.0

.. </legal notes>


**Return:** ``CNM_ReturnTypes.SingleExecutionResult.SUCCESS``: new Container not needed / could be allocated and data was copied
	``CNM_ReturnTypes.SingleExecutionResult.ERROR``: new Container couldn't be allocated, container left unchanged
	``CNM_ReturnTypes.SingleExecutionResult.ABORTED``: NULL object or the list itself was passed
*)
METHOD prepend :CNM_ReturnTypes.SingleExecutionResult
VAR_INPUT
	(*The object to be prepended*)
	object	: CNM_AbstractObject.IObject;
END_VAR
prepend := THIS^.insertObjectAt(index := 0, object := object);
END_METHOD

(*

## Short summary

This method adds all elements of the given collection to the start of this list. 
The order is given by the default iterator of the given collection.
If the collection to prepend is null or contains no element, list is unchanged.

.. <legal notes>

legal notes
=================
| SPDX-FileCopyrightText: © 2025 ekvip automation GmbH <info@ekvip.de>
| SPDX-License-Identifier: Apache-2.0
| For details check: Apache-2.0_

.. _Apache-2.0: https://www.apache.org/licenses/LICENSE-2.0

.. </legal notes>


**Return:** ``CNM_ReturnTypes.SingleExecutionResult.SUCCESS``: prepend was successful
	``CNM_ReturnTypes.SingleExecutionResult.ERROR``: collection to prepend didn't fit in old container, and new container couldn't be allocated
	``CNM_ReturnTypes.SingleExecutionResult.ABORTED``: NULL object or this arraylist was passed
	
*)
METHOD prependCollection :CNM_ReturnTypes.SingleExecutionResult
VAR_INPUT
	(*The collection to be prepended*)
	collectionToPrepend		:CNM_CollectionInterfaces.ICollection;
END_VAR
VAR
	currentIndex 			:UDINT;
	currentObject 			:CNM_AbstractObject.IObject;
	offset 					:__UXINT;
	iterator				:CNM_CollectionInterfaces.IIterator;
	newContainer			:POINTER TO CNM_AbstractObject.IObject;
	arrayListToPrepend		:POINTER TO ArrayList;
	newContainerSize		:UDINT;
END_VAR
VAR CONSTANT
	REGISTER_SIZE :UDINT := SIZEOF(__XWORD);
END_VAR
prependCollection := CNM_ReturnTypes.SingleExecutionResult.ABORTED;
RETURN(THIS^.isObjectNull(collectionToPrepend) OR_ELSE THIS^.isEqual(collectionToPrepend));
prependCollection := CNM_ReturnTypes.SingleExecutionResult.SUCCESS;
RETURN (collectionToPrepend.size = 0);
prependCollection := CNM_ReturnTypes.SingleExecutionResult.ERROR;
THIS^.resizingStrategy.getUpscaledCapacity(requestedSize := THIS^.size + collectionToPrepend.size, currentCapacity := THIS^.currentContainerCapacity, newCapacity => newContainerSize);
newContainer := __NEW(__XWORD, newContainerSize);
RETURN(newContainer = 0);
IF (Tc2_System.MEMMOVE(ADR(newContainer[collectionToPrepend.size]), THIS^.container, THIS^.size * REGISTER_SIZE) = 0) THEN
	__DELETE(newContainer);
	RETURN;
END_IF
IF (__QUERYPOINTER(collectionToPrepend, arrayListToPrepend)) THEN
	IF (Tc2_System.MEMMOVE(newContainer, arrayListToPrepend^.container, collectionToPrepend.size*REGISTER_SIZE) = 0) THEN
		__DELETE(newContainer);
		RETURN;
	END_IF
ELSE
	IF (collectionToPrepend.createNewIterator(iterator => iterator) <> CNM_ReturnTypes.SingleExecutionResult.SUCCESS) THEN
		__DELETE(newContainer); 
		RETURN;
	END_IF
	
	iterator.iterate(execute := FALSE);
	WHILE (
		iterator.iterate(execute := TRUE, object => currentObject) 
		= CNM_ReturnTypes.SingleExecutionState.BUSY
	) DO
		newContainer[currentIndex] := currentObject;
		currentIndex := (currentIndex + 1);
	END_WHILE
	iterator.destruct();
	IF (currentIndex < collectionToPrepend.size) THEN
		__DELETE(newContainer); 
		RETURN;
	END_IF
END_IF
__DELETE(THIS^.container);
THIS^.container := newContainer;
THIS^.currentContainerCapacity := newContainerSize;
THIS^.incrementSize(collectionToPrepend.size);
THIS^.announceListChange();
prependCollection := CNM_ReturnTypes.SingleExecutionResult.SUCCESS;
END_METHOD

(*

## Short summary

This method removes the first instance of the given object from the list.
Passing a null object leaves the list unchanged.

.. <legal notes>

legal notes
=================
| SPDX-FileCopyrightText: © 2022 ekvip automation GmbH <info@ekvip.de>
| SPDX-License-Identifier: Apache-2.0
| For details check: Apache-2.0_

.. _Apache-2.0: https://www.apache.org/licenses/LICENSE-2.0

.. </legal notes>



*)
METHOD remove
VAR_INPUT
	(*The object to be removed from the list*)
	object	:CNM_AbstractObject.IObject;
END_VAR
VAR
	index :UDINT;
END_VAR
IF(THIS^.getIndexOf(object, index => index) = CNM_ReturnTypes.SingleExecutionResult.SUCCESS)THEN
	THIS^.removeObjectAt(index);
END_IF
END_METHOD

(*

## Short summary

This method removes the element at the given index from the list (does not destruct it!).
Elements right from the object are shifted to close the gap.

.. <legal notes>

legal notes
=================
| SPDX-FileCopyrightText: © 2022 ekvip automation GmbH <info@ekvip.de>
| SPDX-License-Identifier: Apache-2.0
| For details check: Apache-2.0_

.. _Apache-2.0: https://www.apache.org/licenses/LICENSE-2.0

.. </legal notes>


**Return:** ``CNM_ReturnTypes.SingleExecutionResult.SUCCESS``: remove was successful
	``CNM_ReturnTypes.SingleExecutionResult.ERROR``: index out of bounds

*)
METHOD removeObjectAt :CNM_ReturnTypes.SingleExecutionResult
VAR_INPUT
	(*the index to remove the object from*)
	index	:UDINT;
END_VAR
VAR_OUTPUT
	(*the removed object*)
	object :CNM_AbstractObject.IObject;
END_VAR
VAR CONSTANT
	NULL_REFERENCE :__XWORD := 0;
END_VAR
removeObjectAt := CNM_ReturnTypes.SingleExecutionResult.ERROR;
RETURN (index >= THIS^.size);

removeObjectAt := CNM_ReturnTypes.SingleExecutionResult.SUCCESS;
THIS^.getObjectAt(index := index, object => object);
//return from leftShiftObjects unconsiderd as lack of memory isn't an error for remove
THIS^.leftShiftObjects(index+1);
THIS^.decrementSize();
THIS^.downscaleContainer();
THIS^.announceListChange();
END_METHOD

(*

## Short summary

This method replaces the object inside the collection at the given index with the given object.

Replacing with NULL does not affect the list.

.. <legal notes>

legal notes
=================
| SPDX-FileCopyrightText: © 2022 ekvip automation GmbH <info@ekvip.de>
| SPDX-License-Identifier: Apache-2.0
| For details check: Apache-2.0_

.. _Apache-2.0: https://www.apache.org/licenses/LICENSE-2.0

.. </legal notes>


**Return:** ``CNM_ReturnTypes.SingleExecutionResult.SUCCESS``: index was valid and object at index replaced with given object
	``CNM_ReturnTypes.SingleExecutionResult.ERROR``: index was invalid or object NULL, nothing changed


*)

METHOD replaceObjectAt :CNM_ReturnTypes.SingleExecutionResult
VAR_INPUT	
	(*the index to replace the object at*)
	index :UDINT;
	(*the object to be at this index instead*)
	withObject :CNM_AbstractObject.IObject;
END_VAR
replaceObjectAt := CNM_ReturnTypes.SingleExecutionResult.ERROR;
RETURN (index >= THIS^.size);

IF (THIS^.isObjectValid(withObject)) THEN
	THIS^.container[index] := withObject;
	replaceObjectAt := CNM_ReturnTypes.SingleExecutionResult.SUCCESS;
	THIS^.announceListChange();
END_IF
END_METHOD

(*

## Short summary

This property can be used to inject a customized resizing strategy for arrays and containers. 
The getter returns the currently used strategy as a fluent interface.
If no custom strategy is set, a default strategy will be used. 

.. <legal notes>

legal notes
=================
| SPDX-FileCopyrightText: © 2025 ekvip automation GmbH <info@ekvip.de>
| SPDX-License-Identifier: Apache-2.0
| For details check: Apache-2.0_

.. _Apache-2.0: https://www.apache.org/licenses/LICENSE-2.0

.. </legal notes>

*)

PROPERTY resizingStrategy : CNM_CollectionInterfaces.IResizingStrategy
GET
VAR_STAT
	defaultStrategy :CubicRootResizing;
END_VAR
IF THIS^.isObjectValid(THIS^.injectedResizingStrategy) THEN
	resizingStrategy := THIS^.injectedResizingStrategy;
ELSE
	resizingStrategy := defaultStrategy;
END_IF
END_GET
SET
THIS^.injectedResizingStrategy := resizingStrategy;
END_SET
END_PROPERTY

(*

## Short summary

This method shifts all ojects in the container from startIndex to size - 1 to the right.
Ensure that the container has sufficient space to perform the shift, otherwise it will return ERROR.
rightShift(0) : A B C D -> _ A B C D


.. <legal notes>

legal notes
=================
| SPDX-FileCopyrightText: © 2025 ekvip automation GmbH <info@ekvip.de>
| SPDX-License-Identifier: Apache-2.0
| For details check: Apache-2.0_

.. _Apache-2.0: https://www.apache.org/licenses/LICENSE-2.0

.. </legal notes>


**Return:** ``CNM_ReturnTypes.SingleExecutionResult.SUCCESS``: rightshift was successful
	``CNM_ReturnTypes.SingleExecutionResult.ERROR``: startindex behind last object or not enough space inside the container. 

*)

METHOD PROTECTED rightShiftObjects :CNM_ReturnTypes.SingleExecutionResult
VAR_INPUT
	(* the index of the first element which will be shifted *)
	startIndex 	:UDINT;
	distance 	:UDINT := 1;
END_VAR
VAR
	offset 				:UDINT;
	length 				:UDINT;
	objectsToShift		:UDINT;
END_VAR
VAR CONSTANT
	IS_NOT_REFERENCED 	:USINT := 0;
	REGISTER_SIZE :UDINT := SIZEOF(__XWORD);
END_VAR
rightShiftObjects := CNM_ReturnTypes.SingleExecutionResult.ERROR;
RETURN((startIndex > THIS^.size) OR_ELSE (distance > THIS^.currentContainerCapacity - THIS^.size ));
rightShiftObjects := CNM_ReturnTypes.SingleExecutionResult.SUCCESS;
objectsToShift := THIS^.size - startIndex;
RETURN(objectsToShift = 0);
Tc2_System.MEMMOVE(ADR(THIS^.container[startIndex+distance]), ADR(THIS^.container[startIndex]), objectsToShift * REGISTER_SIZE);
Tc2_System.MEMSET(ADR(THIS^.container[startIndex]), IS_NOT_REFERENCED, distance * REGISTER_SIZE);
END_METHOD

(*

## Short summary

This method can replace the default sorter for a custom one. Check ``IListSorter`` and ``IArrayListSorter``

.. warning
	If the a dynamic instance of an injected sorter already exists, it will be destructed.
	
.. warning
	If the injected sorter was created dynamically,
	it will be automatically destruced within the destruct context of THIS list.
	
.. <legal notes>

legal notes
=================
| SPDX-FileCopyrightText: © 2025 ekvip automation GmbH <info@ekvip.de>
| SPDX-License-Identifier: Apache-2.0
| For details check: Apache-2.0_

.. _Apache-2.0: https://www.apache.org/licenses/LICENSE-2.0

.. </legal notes>


**Return:** ``THIS`` :``ISortable``

*)
METHOD setSorter :CNM_CollectionInterfaces.ISortable
VAR_INPUT
	(*The instance of the sorter to be used to sort the list*)
	sorter	:CNM_CollectionInterfaces.IArrayListSorter;
END_VAR
THIS^.injectedSorter := sorter;
setSorter := THIS^.sort;
END_METHOD

PROPERTY PROTECTED sorter :CNM_CollectionInterfaces.IArrayListSorter
GET
VAR_INST
	instSorter :ArrayListShellSorter;
END_VAR
IF(THIS^.isObjectValid(THIS^.injectedSorter))THEN
	sorter := THIS^.injectedSorter;
ELSE
	sorter := instSorter;
END_IF
END_GET
END_PROPERTY

METHOD INTERNAL sorting : CNM_ReturnTypes.SingleExecutionState
VAR_INPUT
	execute :BOOL;
	order :SortingOrder;
	(*Optional: the comparator that should be used for the sort. Must not be changed while sort is in process*)
	comparator	: CNM_CollectionInterfaces.CNM_AbstractObject.IComparator := 0;
END_VAR
CASE order OF
SortingOrder.ASCENDING:
	sorting := THIS^.sorter.sort(
		execute := execute, 
		size := THIS^.size, 
		comparator := comparator, 
		container := THIS^.container, 
		currentListVersion := THIS^.changesToCollection
	);

SortingOrder.DESCENDING:
	sorting	:= THIS^.sorter.inverseSort(
		execute := execute, 
		size := THIS^.size, 
		container := THIS^.container, 
		currentListVersion := THIS^.changesToCollection
	);
	
END_CASE
END_METHOD

(*

## Short summary

This method increases the container to have at least ``space`` more capacity.

.. <legal notes>

legal notes
=================
| SPDX-FileCopyrightText: © 2025 ekvip automation GmbH <info@ekvip.de>
| SPDX-License-Identifier: Apache-2.0
| For details check: Apache-2.0_

.. _Apache-2.0: https://www.apache.org/licenses/LICENSE-2.0

.. </legal notes>


**Return:** ``CNM_ReturnTypes.SingleExecutionResult.SUCCESS``: new container could be allocated and data was transferd
	``CNM_ReturnTypes.SingleExecutionResult.ERROR``: allocation of new container failed

*)

{info 'add logging if allocation fails'}

METHOD PROTECTED upscaleContainer :CNM_ReturnTypes.SingleExecutionResult
VAR_INPUT
	(*The amount of storagecapacity that should be added*)
	space 					:UDINT;
END_VAR
VAR
	newContainer			:POINTER TO CNM_AbstractObject.IObject;
	lastContainerCapacity	:UDINT;
	newContainerCapacity	:UDINT;
END_VAR
lastContainerCapacity := THIS^.currentContainerCapacity;

IF THIS^.resizingStrategy.getUpscaledCapacity(
		requestedSize := THIS^.size + space,
		currentCapacity := THIS^.currentContainerCapacity,
		newCapacity => newContainerCapacity
	)
THEN
	newContainer := __NEW(__XWORD, newContainerCapacity);
	IF (newContainer <> 0) THEN
		IF (THIS^.size > 0) AND_THEN (THIS^.container <> 0) THEN
			Tc2_System.MEMMOVE(newContainer, THIS^.container, THIS^.size * SIZEOF(__XWORD));
			__DELETE(THIS^.container);
		END_IF;
		THIS^.container := newContainer;
		upscaleContainer := CNM_ReturnTypes.SingleExecutionResult.SUCCESS;
		THIS^.currentContainerCapacity := newContainerCapacity;
	ELSE
		THIS^.currentContainerCapacity := lastContainerCapacity;
		upscaleContainer := CNM_ReturnTypes.SingleExecutionResult.ERROR;
	END_IF
ELSE 
	upscaleContainer := CNM_ReturnTypes.SingleExecutionResult.SUCCESS;
END_IF
END_METHOD

END_FUNCTION_BLOCK

// ---- Lists/classes/AbstractList.TcPOU
(*

## Short summary

An abstract class to implement methods which are not dependent on the data structure.

.. <legal notes>

legal notes
=================
| SPDX-FileCopyrightText: © 2024 ekvip automation GmbH <info@ekvip.de>
| SPDX-License-Identifier: Apache-2.0
| For details check: Apache-2.0_

.. _Apache-2.0: https://www.apache.org/licenses/LICENSE-2.0

.. </legal notes>



*)
FUNCTION_BLOCK ABSTRACT AbstractList EXTENDS AbstractCollection IMPLEMENTS CNM_CollectionInterfaces.IList, IListHelpers

(*

## Short summary

This method adds the given CNM_AbstractObject.IObject to the end of the list.
**Example:** 
Given a list that looks like this: (Head->) A B C (<- End),
calling append(D) on this list will place the D at the and,
making it the new End: (Head->) A B C D(<- End)

.. <legal notes>

legal notes
=================
| SPDX-FileCopyrightText: © 2022 ekvip automation GmbH <info@ekvip.de>
| SPDX-License-Identifier: Apache-2.0
| For details check: Apache-2.0_

.. _Apache-2.0: https://www.apache.org/licenses/LICENSE-2.0

.. </legal notes>



*)

METHOD ABSTRACT append :CNM_ReturnTypes.SingleExecutionResult
VAR_INPUT
	(*The object to be appended*)
	object		:CNM_AbstractObject.IObject;
END_VAR
END_METHOD

(*

## Short summary

This method adds all elements of the given collection to the end of this list.
**Example:**
For the list1: A B C and list2: D E F will be after ```list1.appendCollection(list2)```:
A B C D E F. Notice the elements are still in the same order they where befor on each subsection.

.. <legal notes>

legal notes
=================
| SPDX-FileCopyrightText: © 2022 ekvip automation GmbH <info@ekvip.de>
| SPDX-License-Identifier: Apache-2.0
| For details check: Apache-2.0_

.. _Apache-2.0: https://www.apache.org/licenses/LICENSE-2.0

.. </legal notes>


**Return:** ``CNM_ReturnTypes.SingleExecutionResult.SUCCESS``: new Container not needed / could be allocated and data was copied
	``CNM_ReturnTypes.SingleExecutionResult.ERROR``: new Container couldn't be allocated, container left unchanged
	``CNM_ReturnTypes.SingleExecutionResult.ABORTED``: NULL object or the list itself was passed

*)

METHOD ABSTRACT appendCollection :CNM_ReturnTypes.SingleExecutionResult
VAR_INPUT
	(*The collection to be appended*)
	collectionToAppend :CNM_CollectionInterfaces.ICollection;
END_VAR
END_METHOD

(*

## Short summary

This abstract property returns the class name of the concrete object, 
which is useful to check the class name for ``__DELETE``.

.. <legal notes>

legal notes
=================
| SPDX-FileCopyrightText: © 2022 ekvip automation GmbH <info@ekvip.de>
| SPDX-License-Identifier: Apache-2.0
| For details check: Apache-2.0_

.. _Apache-2.0: https://www.apache.org/licenses/LICENSE-2.0

.. </legal notes>

*)
PROPERTY ABSTRACT className : CNM_AbstractObject.ClassName
GET
END_GET
END_PROPERTY

(*

## Short summary

This property returns the last object in the first and removes it from the list. Can be seen as opposite of prepend.
**Example:**
On a list: (Head -->) A B C, list.dequeue will return A.
**Example 2:**
If you call prepend(x), a dequeue right after will return x.

.. <legal notes>

legal notes
=================
| SPDX-FileCopyrightText: © 2022 ekvip automation GmbH <info@ekvip.de>
| SPDX-License-Identifier: Apache-2.0
| For details check: Apache-2.0_

.. _Apache-2.0: https://www.apache.org/licenses/LICENSE-2.0

.. </legal notes>

*)

METHOD ABSTRACT dequeue :CNM_AbstractObject.IObject
END_METHOD

METHOD INTERNAL ABSTRACT instantSorting : CNM_ReturnTypes.SingleExecutionResult
VAR_INPUT
	order :SortingOrder;
	(*Optional: the comparator that should be used for the sort. Must not be changed while sort is in process*)
	comparator	: CNM_CollectionInterfaces.CNM_AbstractObject.IComparator := 0;
END_VAR
END_METHOD

(*

## Short summary

Inverts the order of the elements inside the object. Does not apply any kind of sorting, only reverses.

.. <legal notes>

legal notes
=================
| SPDX-FileCopyrightText: © 2022 ekvip automation GmbH <info@ekvip.de>
| SPDX-License-Identifier: Apache-2.0
| For details check: Apache-2.0_

.. _Apache-2.0: https://www.apache.org/licenses/LICENSE-2.0

.. </legal notes>



*)

METHOD ABSTRACT invert
END_METHOD

PROPERTY INTERNAL listChangeIndex : __XWORD
GET
listChangeIndex := THIS^.changesToCollection;
END_GET
SET
THIS^.changesToCollection := listChangeIndex;
END_SET
END_PROPERTY

(*

## Short summary

This property returns the last object in the list and removes it from the list. Can be seen as opposite of append.
**Example:**
On a list: (Head -->) A B C, list.pop will return C.
**Example 2:**
If you call append(x), a pop right after will return x.
May return a null pointer if list is empty

.. <legal notes>

legal notes
=================
| SPDX-FileCopyrightText: © 2022 ekvip automation GmbH <info@ekvip.de>
| SPDX-License-Identifier: Apache-2.0
| For details check: Apache-2.0_

.. _Apache-2.0: https://www.apache.org/licenses/LICENSE-2.0

.. </legal notes>

*)

METHOD ABSTRACT pop :CNM_AbstractObject.IObject
END_METHOD

(*

## Short summary

This method adds the given obejct to the end of the list.
**Example:** 
Given a list that looks like this: (Head->) A B C (<- End),
calling prepend(D) on this list will place the D at start,
making it the new Head: (Head->) D A B C (<- End)

.. <legal notes>

legal notes
=================
| SPDX-FileCopyrightText: © 2022 ekvip automation GmbH <info@ekvip.de>
| SPDX-License-Identifier: Apache-2.0
| For details check: Apache-2.0_

.. _Apache-2.0: https://www.apache.org/licenses/LICENSE-2.0

.. </legal notes>


**Return:** ``CNM_ReturnTypes.SingleExecutionResult.SUCCESS``: new Container not needed / could be allocated and data was copied
	``CNM_ReturnTypes.SingleExecutionResult.ERROR``: new Container couldn't be allocated, container left unchanged
	``CNM_ReturnTypes.SingleExecutionResult.ABORTED``: NULL object or the list itself was passed
	
*)

METHOD ABSTRACT prepend :CNM_ReturnTypes.SingleExecutionResult
VAR_INPUT
	(*The object to be prepended*)
	object	:CNM_AbstractObject.IObject;
END_VAR
END_METHOD

(*

## Short summary

This method adds all elements of the given collection to the start of this list. 
**Example:**
For the list1: A B C and list2: D E F will be after ```list1.prependCollection(list2)```:
D E F A B C. Notice the elements are still in the same order they where befor on each subsection.

.. <legal notes>

legal notes
=================
| SPDX-FileCopyrightText: © 2022 ekvip automation GmbH <info@ekvip.de>
| SPDX-License-Identifier: Apache-2.0
| For details check: Apache-2.0_

.. _Apache-2.0: https://www.apache.org/licenses/LICENSE-2.0

.. </legal notes>


**Return:** ``CNM_ReturnTypes.SingleExecutionResult.SUCCESS``: prepend was successful
	``CNM_ReturnTypes.SingleExecutionResult.ERROR``: collection to prepend didn't fit in old container, and new container couldn't be allocated
	``CNM_ReturnTypes.SingleExecutionResult.ABORTED``: NULL object or this arraylist was passed
	
*)

METHOD ABSTRACT prependCollection :CNM_ReturnTypes.SingleExecutionResult
VAR_INPUT
	(*The collection to be prepended*)
	collectionToPrepend :CNM_CollectionInterfaces.ICollection;
END_VAR
END_METHOD

(*

## Short summary

This method removes the first instance of the given object from the list.
Compares objects with hash value.
For example a Linked List: A B C A A D after remove(A) becomes: B C A A D

.. <legal notes>

legal notes
=================
| SPDX-FileCopyrightText: © 2022 ekvip automation GmbH <info@ekvip.de>
| SPDX-License-Identifier: Apache-2.0
| For details check: Apache-2.0_

.. _Apache-2.0: https://www.apache.org/licenses/LICENSE-2.0

.. </legal notes>



*)

METHOD ABSTRACT remove
VAR_INPUT
	(*The object to be removed from the list*)
	object		:CNM_AbstractObject.IObject;
END_VAR
END_METHOD

(*

## Short summary

This property returns strategies to sort the list in a desired order.

.. <legal notes>

legal notes
=================
| SPDX-FileCopyrightText: © 2024 ekvip automation GmbH <info@ekvip.de>
| SPDX-License-Identifier: Apache-2.0
| For details check: Apache-2.0_

.. _Apache-2.0: https://www.apache.org/licenses/LICENSE-2.0

.. </legal notes>

*)

PROPERTY sort : CNM_CollectionInterfaces.ISortable
GET
VAR_INST
	sortStrategy	:SortingStrategyExecutor(THIS^);
END_VAR
sort := sortStrategy;
END_GET
END_PROPERTY

METHOD INTERNAL ABSTRACT sorting : CNM_ReturnTypes.SingleExecutionState
VAR_INPUT
	execute :BOOL;
	order :SortingOrder;
	(*Optional: the comparator that should be used for the sort. Must not be changed while sort is in process*)
	comparator	: CNM_CollectionInterfaces.CNM_AbstractObject.IComparator := 0;
END_VAR
END_METHOD

END_FUNCTION_BLOCK

// ---- Collection/classes/AbstractCollection.TcPOU
(*

## Short summary

An abstract class to implement the basic datastructure independend collection functionality for use in 
other Collections.

.. <legal notes>

legal notes
=================
| SPDX-FileCopyrightText: © 2022 ekvip automation GmbH <info@ekvip.de>
| SPDX-License-Identifier: Apache-2.0
| For details check: Apache-2.0_

.. _Apache-2.0: https://www.apache.org/licenses/LICENSE-2.0

.. </legal notes>



*)

FUNCTION_BLOCK ABSTRACT AbstractCollection EXTENDS AbstractDisposableContainer IMPLEMENTS CNM_CollectionInterfaces.ICollection
VAR
	(*the amount of objects in the collection*)
	collectionSize 		:UDINT;
	(*counter that increases on every collection change*)
	changesToCollection :__XWORD;
END_VAR
VAR_STAT
	collectionFactory 	:CollectionFactory();
END_VAR

(*

## Short summary

This method clears/deletes all clearable data from this object.
**Example:**
A list: 1 2 3 after ```list.clear()``` will have no remaining items, isEmpty = true.

.. <legal notes>

legal notes
=================
| SPDX-FileCopyrightText: © 2022 ekvip automation GmbH <info@ekvip.de>
| SPDX-License-Identifier: Apache-2.0
| For details check: Apache-2.0_

.. _Apache-2.0: https://www.apache.org/licenses/LICENSE-2.0

.. </legal notes>



*)

METHOD ABSTRACT clear
END_METHOD

(*

## Short summary

This method compares a foreign object with the own one, this is needed for sort orders.
The abstract class evaluates every object that is NULL as greater, and all other objects as equal. 

.. <legal notes>

legal notes
=================
| SPDX-FileCopyrightText: © 2022 ekvip automation GmbH <info@ekvip.de>
| SPDX-License-Identifier: Apache-2.0
| For details check: Apache-2.0_

.. _Apache-2.0: https://www.apache.org/licenses/LICENSE-2.0

.. </legal notes>


**Return:** ``SMALLER``: ``THIS`` precedes in order,
	``EQUAL``: ``THIS`` and ``object`` at the same position in order,
	``GREATER``: ``THIS`` is after in order.
	Checkout :``CNM_CollectionInterfaces.ComparationResult``.

*)
METHOD compareTo :CNM_ReturnTypes.ComparationResult
VAR_INPUT
	(*the object to be compared to*)
	object	:CNM_CollectionInterfaces.CNM_AbstractObject.IObject;
END_VAR
VAR
	collection :CNM_CollectionInterfaces.ICollection;
END_VAR
IF (THIS^.isObjectNull(object)) THEN
	compareTo := CNM_ReturnTypes.ComparationResult.GREATER;
ELSE
	compareTo := CNM_ReturnTypes.ComparationResult.EQUAL;
	IF(__QUERYINTERFACE(object, collection)) THEN
		IF(collection.size < THIS^.size) THEN
			compareTo := CNM_ReturnTypes.ComparationResult.GREATER;
		ELSIF(collection.size > THIS^.size) THEN
			compareTo := CNM_ReturnTypes.ComparationResult.SMALLER;			
		END_IF
	END_IF
END_IF
END_METHOD

(*

## Short summary

This method checks if a given object is contained in the collection. 
The object is inside if the collection contains an object where the compareTo returns EQUAL.

.. <legal notes>

legal notes
=================
| SPDX-FileCopyrightText: © 2022 ekvip automation GmbH <info@ekvip.de>
| SPDX-License-Identifier: Apache-2.0
| For details check: Apache-2.0_

.. _Apache-2.0: https://www.apache.org/licenses/LICENSE-2.0

.. </legal notes>


**Return:** ``FALSE``: collection does not contain an equal object
    ``TRUE``: collection does contain an equal object

*)

METHOD containsEqualObject :BOOL
VAR_INPUT
	(*the object to be checked if it exists inside the collection*)
	object	:CNM_AbstractObject.IObject;
END_VAR
VAR
	currentObj :CNM_AbstractObject.IObject;
END_VAR
containsEqualObject := FALSE;
RETURN(NOT THIS^.isObjectValid(object));
THIS^.iterate(execute := FALSE);
WHILE (THIS^.iterate(execute := TRUE, object => currentObj) = CNM_ReturnTypes.SingleExecutionState.BUSY) DO
	IF (object.compareTo(currentObj) = CNM_ReturnTypes.ComparationResult.EQUAL) THEN
		containsEqualObject := TRUE;
		RETURN;
	END_IF
END_WHILE
END_METHOD

(*

## Short summary

This method checks if a given object is contained in the collection. 
The object is inside if the collection contains an object for that isEqual retuns true.

.. <legal notes>

legal notes
=================
| SPDX-FileCopyrightText: © 2022 ekvip automation GmbH <info@ekvip.de>
| SPDX-License-Identifier: Apache-2.0
| For details check: Apache-2.0_

.. _Apache-2.0: https://www.apache.org/licenses/LICENSE-2.0

.. </legal notes>


**Return:** ``FALSE``: collection does not contain given object,
    ``TRUE``: collection does contain given object

*)

METHOD containsObject :BOOL
VAR_INPUT
	(*the object to be checked if it exists inside the collection*)
	object	:CNM_AbstractObject.IObject;
END_VAR
VAR
	currentObj :CNM_AbstractObject.IObject;
END_VAR
containsObject := FALSE;
RETURN(NOT THIS^.isObjectValid(object));
THIS^.iterate(execute := FALSE);
WHILE(THIS^.iterate(execute := TRUE, object => currentObj) = CNM_ReturnTypes.SingleExecutionState.BUSY)DO
	IF(object.isEqual(currentObj))THEN
		containsObject := TRUE;
		RETURN;
	END_IF
END_WHILE
END_METHOD

(*

## Short summary

This method returns a NEW Iterator instance which can iterate the collection.
These iterators can be used parallel independend of each other on the same collection.

**Warning:**
The returned Iterator was created using the __NEW operator and must be destructed to avoid memory leaks!



.. <legal notes>

legal notes
=================
| SPDX-FileCopyrightText: © 2024 ekvip automation GmbH <info@ekvip.de>
| SPDX-License-Identifier: Apache-2.0
| For details check: Apache-2.0_

.. _Apache-2.0: https://www.apache.org/licenses/LICENSE-2.0

.. </legal notes>



*)

METHOD ABSTRACT createNewIterator :CNM_ReturnTypes.SingleExecutionResult
VAR_OUTPUT
	(*The new created iterator or null if allocation fails *)
	iterator :CNM_CollectionInterfaces.IIterator;
END_VAR
END_METHOD

(*

## Short summary

This property returns strategies to loop through the collection and apply actions to all objects contained.

.. <legal notes>

legal notes
=================
| SPDX-FileCopyrightText: © 2024 ekvip automation GmbH <info@ekvip.de>
| SPDX-License-Identifier: Apache-2.0
| For details check: Apache-2.0_

.. _Apache-2.0: https://www.apache.org/licenses/LICENSE-2.0

.. </legal notes>

*)

PROPERTY forEach :CNM_CollectionInterfaces.IForEachStrategy
GET
VAR_INST
	executor : ForEachStrategyExecutor(THIS^);
END_VAR
forEach := executor;
END_GET
END_PROPERTY

(*

## Short summary

This property returns ``TRUE`` if the collection has any element.

.. <legal notes>

legal notes
=================
| SPDX-FileCopyrightText: © 2022 ekvip automation GmbH <info@ekvip.de>
| SPDX-License-Identifier: Apache-2.0
| For details check: Apache-2.0_

.. _Apache-2.0: https://www.apache.org/licenses/LICENSE-2.0

.. </legal notes>

*)

PROPERTY FINAL hasElement :BOOL
GET
hasElement := (THIS^.size > 0);
END_GET
END_PROPERTY

(*

## Short summary

This property returns ``TRUE`` if the collection is empty.

.. <legal notes>

legal notes
=================
| SPDX-FileCopyrightText: © 2022 ekvip automation GmbH <info@ekvip.de>
| SPDX-License-Identifier: Apache-2.0
| For details check: Apache-2.0_

.. _Apache-2.0: https://www.apache.org/licenses/LICENSE-2.0

.. </legal notes>

*)

PROPERTY FINAL isEmpty :BOOL
GET
isEmpty := (THIS^.size = 0);
END_GET
END_PROPERTY

(*

## Short summary

This method returns the next object in the iteration and returns an execution state.
**Example:**
You have a list: 1 2 3
the first iterate call will return CNM_ReturnTypes.BUSY and object = 1
the second iterate call will return CNM_ReturnTypes.BUSY and object = 2
the third iterate call will return CNM_ReturnTypes.BUSY and object = 3
the fourth iterate call will return CNM_ReturnTypes.SUCCESS and object = null;

.. <legal notes>

legal notes
=================
| SPDX-FileCopyrightText: © 2022 ekvip automation GmbH <info@ekvip.de>
| SPDX-License-Identifier: Apache-2.0
| For details check: Apache-2.0_

.. _Apache-2.0: https://www.apache.org/licenses/LICENSE-2.0

.. </legal notes>


**Return:** ``SUCCESS``: if last object from collection was already returned,
    ``ABORTED``: execute has a falling edge during iterate,
    ``BUSY``: When iterate had rising edge on execute and not all objects had been returned yet,
    ``IDLE``: iterate wasn't started yet,
	``ERROR``: error occured during iteration 

*)

METHOD PROTECTED ABSTRACT iterate :CNM_ReturnTypes.SingleExecutionState
VAR_INPUT
	(*Indicates if the iteration should be executed or resetted*) 
	execute	:BOOL;
END_VAR
VAR_OUTPUT
	(*The current Object of the Iteration*)
	object	:CNM_AbstractObject.IObject;
END_VAR
END_METHOD

(*

## Short summary

This property returns the number of elements inside this collection.

.. <legal notes>

legal notes
=================
| SPDX-FileCopyrightText: © 2022 ekvip automation GmbH <info@ekvip.de>
| SPDX-License-Identifier: Apache-2.0
| For details check: Apache-2.0_

.. _Apache-2.0: https://www.apache.org/licenses/LICENSE-2.0

.. </legal notes>

*)

PROPERTY FINAL size :UDINT
GET
size := THIS^.collectionSize;
END_GET
END_PROPERTY

END_FUNCTION_BLOCK

// ---- Factories/classes/CollectionFactory.TcPOU
(*

## Short summary

Class that provides factory methods for new collection instances.

.. <legal notes>

legal notes
=================
| SPDX-FileCopyrightText: © 2022 ekvip automation GmbH <info@ekvip.de>
| SPDX-License-Identifier: Apache-2.0
| For details check: Apache-2.0_

.. _Apache-2.0: https://www.apache.org/licenses/LICENSE-2.0

.. </legal notes>



*)
FUNCTION_BLOCK CollectionFactory EXTENDS CNM_AbstractObject.Object IMPLEMENTS CNM_CollectionInterfaces.ICollectionFactory

(*

## Short summary

This abstract property returns the class name of the concrete object, 
which is useful to check the class name for ``__DELETE``.

.. <legal notes>

legal notes
=================
| SPDX-FileCopyrightText: © 2022 ekvip automation GmbH <info@ekvip.de>
| SPDX-License-Identifier: Apache-2.0
| For details check: Apache-2.0_

.. _Apache-2.0: https://www.apache.org/licenses/LICENSE-2.0

.. </legal notes>

*)
PROPERTY className : CNM_AbstractObject.ClassName
GET
className := 'CNM_Collections.CollectionFactory';
END_GET
END_PROPERTY

(*

## Short summary

This method is used to create a new instance
of the object which has the same internal state as the object.
If the object is a container class, the references to the content objects
are not cloned for this there is the method `ICloneable.deepClone`.

If an object does not support cloning the return value is
``CNM_ReturnTypes.CloneResult.CLONE_IS_NOT_SUPPORTED``.

If there is not enough memory or the cloning fails because the
attribute enable dynamic creation was forgotten the return value is 
``CNM_ReturnTypes.CloneResult.FAILED``.

Only if the return value is ``CNM_ReturnTypes.CloneResult.SUCCESS``
the output ``clonedObject`` points to the new object
otherwise ``clonedObject`` is NULL.  

**Attention:** 
	For derivations: **If a derived class needs ``clone`` this method must be overwritten.**
	and don't forget the attribute ``{attribute 'enable_dynamic_creation'}``  

.. <legal notes>

legal notes
=================
| SPDX-FileCopyrightText: © 2022 ekvip automation GmbH <info@ekvip.de>
| SPDX-License-Identifier: Apache-2.0
| For details check: Apache-2.0_

.. _Apache-2.0: https://www.apache.org/licenses/LICENSE-2.0

.. </legal notes>


**Return:** ``CNM_ReturnTypes.CloneResult.SUCCESS``: new object clone was created,
	``CNM_ReturnTypes.CloneResult.FAILED``: object clone failed
	``CNM_ReturnTypes.CloneResult.CLONE_IS_NOT_SUPPORTED``: object does not support cloning

*)

METHOD clone :CNM_ReturnTypes.CloneResult
VAR_OUTPUT
	(* new object instance or NULL if somthing went wrong *)
	clonedObject	:CNM_AbstractObject.IObject;
END_VAR
IF (
	Tc2_System.F_CheckMemoryArea(pData := THIS, nSize := SIZEOF(THIS^))
	= Tc2_System.E_TcMemoryArea.Static
) THEN
	clonedObject := THIS^;
	clone := CNM_ReturnTypes.CloneResult.SUCCESS;
ELSE
	clonedObject := 0;
	clone := CNM_ReturnTypes.CloneResult.CLONE_IS_NOT_SUPPORTED;
END_IF
END_METHOD

(*

## Short summary

This method is used to create a new instance
of the object which has the same internal state as the object.
If the object is a container class, the references to the content objects
are cloned too.

If an object does not support cloning the return value is
``CNM_ReturnTypes.CloneResult.CLONE_IS_NOT_SUPPORTED``.

If there is not enough memory or the cloning fails because the
attribute enable dynamic creation was forgotten the return value is 
``CNM_ReturnTypes.CloneResult.FAILED``.
If something goes wrong, then this method must clean up everything
that has been cloned and free the memory again.
**The deepClone either works completely, or not at all**

Only if the return value is ``CNM_ReturnTypes.CloneResult.SUCCESS``
the output ``clonedObject`` points to the new object
otherwise ``clonedObject`` is NULL.  

**Attention:** 
	For derivations: **If a derived class needs ``deepClone`` this method must be overwritten.**
	and don't forget the attribute ``{attribute 'enable_dynamic_creation'}``, even for container content 

.. <legal notes>

legal notes
=================
| SPDX-FileCopyrightText: © 2022 ekvip automation GmbH <info@ekvip.de>
| SPDX-License-Identifier: Apache-2.0
| For details check: Apache-2.0_

.. _Apache-2.0: https://www.apache.org/licenses/LICENSE-2.0

.. </legal notes>


**Return:**``CNM_ReturnTypes.CloneResult.SUCCESS``: new object clone was created,
``CNM_ReturnTypes.CloneResult.FAILED``: object clone failed
``CNM_ReturnTypes.CloneResult.CLONE_IS_NOT_SUPPORTED``: object does not support deep cloning

*)

METHOD deepClone :CNM_ReturnTypes.CloneResult
VAR_OUTPUT
	(* new object instance or NULL if somthing went wrong *)
	clonedObject	:CNM_AbstractObject.IObject;
END_VAR
deepClone := THIS^.clone(clonedObject => clonedObject);
END_METHOD

(*

## Short summary

A method to generate a new ArrayList.

.. <legal notes>

legal notes
=================
| SPDX-FileCopyrightText: © 2022 ekvip automation GmbH <info@ekvip.de>
| SPDX-License-Identifier: Apache-2.0
| For details check: Apache-2.0_

.. _Apache-2.0: https://www.apache.org/licenses/LICENSE-2.0

.. </legal notes>


**Return:** ``SingleExecutionResult.SUCCESS``: allocation succesful, output arrayList contains new list
    ``SingleExecutionResult.ERROR``: error during allocation, output arrayList is NULL

*)

METHOD getNewArrayList :CNM_ReturnTypes.SingleExecutionResult
VAR_OUTPUT
	(* the created array list *)
	arrayList :CNM_CollectionInterfaces.IArrayList;
END_VAR
VAR
	newList	:POINTER TO ArrayList;
END_VAR
getNewArrayList := CNM_ReturnTypes.SingleExecutionResult.ERROR;
newList := __NEW(ArrayList);
IF (newList <> 0) THEN
	arrayList := newList^;
	getNewArrayList := CNM_ReturnTypes.SingleExecutionResult.SUCCESS;	
END_IF
END_METHOD

(*

## Short summary

This method will create a new MergeSorter

.. <legal notes>

legal notes
=================
| SPDX-FileCopyrightText: © 2022 ekvip automation GmbH <info@ekvip.de>
| SPDX-License-Identifier: Apache-2.0
| For details check: Apache-2.0_

.. _Apache-2.0: https://www.apache.org/licenses/LICENSE-2.0

.. </legal notes>


**Return:** ``SingleExecutionResult.SUCCESS``: allocation succesful, output sorter contains new sorter instance
    ``SingleExecutionResult.ERROR``: error during allocation, output sorter is NULL

*)

METHOD getNewArrayListMergeSorter :CNM_ReturnTypes.SingleExecutionResult
VAR_OUTPUT
	(* the created array list merger sorter *)
	sorter :CNM_CollectionInterfaces.IArrayListSorter;
END_VAR
VAR
	newSorter :POINTER TO ArrayListMergeSorter;
END_VAR
getNewArrayListMergeSorter := CNM_ReturnTypes.SingleExecutionResult.ERROR;
newSorter := __NEW(
	ArrayListMergeSorter()
);
IF (newSorter <> 0) THEN
	sorter := newSorter^;
	getNewArrayListMergeSorter := CNM_ReturnTypes.SingleExecutionResult.SUCCESS;
END_IF
END_METHOD

(*

## Short summary

This method will create a new shellsorter that can sort an Arraylist

.. <legal notes>

legal notes
=================
| SPDX-FileCopyrightText: © 2022 ekvip automation GmbH <info@ekvip.de>
| SPDX-License-Identifier: Apache-2.0
| For details check: Apache-2.0_

.. _Apache-2.0: https://www.apache.org/licenses/LICENSE-2.0

.. </legal notes>


**Return:** ``SingleExecutionResult.SUCCESS``: allocation succesful, output sorter contains new sorter instance
    ``SingleExecutionResult.ERROR``: error during allocation, output sorter is NULL
	
*)

METHOD getNewArrayListShellsorter :CNM_ReturnTypes.SingleExecutionResult
VAR_OUTPUT
	(* the created array list shell sorter *)
	sorter :CNM_CollectionInterfaces.IArrayListSorter;
END_VAR
VAR
	newSorter :POINTER TO ArrayListShellSorter;
END_VAR
getNewArrayListShellSorter := CNM_ReturnTypes.SingleExecutionResult.ERROR;
newSorter := __NEW(
	ArrayListShellSorter()
);
IF (newSorter <> 0) THEN
	sorter := newSorter^;
	getNewArrayListShellSorter := CNM_ReturnTypes.SingleExecutionResult.SUCCESS;
END_IF
END_METHOD

(*

## Short summary

This method can be used to dynamically create a __NEW binary balanced search tree.

.. <legal notes>

legal notes
=================
| SPDX-FileCopyrightText: © 2022 ekvip automation GmbH <info@ekvip.de>
| SPDX-License-Identifier: Apache-2.0
| For details check: Apache-2.0_

.. _Apache-2.0: https://www.apache.org/licenses/LICENSE-2.0

.. </legal notes>


**Return:** ``SingleExecutionResult.SUCCESS``: allocation succesful, output tree contains new tree instance
    ``SingleExecutionResult.ERROR``: error during allocation, output tree is NULL

*)

